FUNCTION_BLOCK "Blok_Pracy_Bindownicy"	// FB 35
//Funkcja odpowiada za sterowanie calym procesem bindowania
//Jezeli dane zostaly zmienione w trakcie trwania cyklu to dopiero w czasie 
//nowego 
//cyklu zostana przyjete.
//
//
//
VERSION : 0.1
VAR_INPUT
  i_Marka_Bezpieczenstwa : BOOL ;
  i_Auto_Reczny : BOOL ;
  i_Bindownica_Auto : BOOL ;
  i_Start_Cyklu_Auto : BOOL ;
  i_Reset_Bledu_Cyklu : BOOL ;
  i_Reset_Cyklu : BOOL ;	//Sprowadza funkcje do poczatku
  i_Pozycjonuj_Palete : BOOL ;
  i_TP_Wiazanie_0_st : BOOL ;
  i_TP_Wiazanie_90_st : BOOL ;
  i_TP_Wiazanie_180_st : BOOL ;
  i_TP_Wiazanie_270_st : BOOL ;
  i_TP_Pozycjonowanie : BOOL ;
  i_s_Zez_Rolki : BOOL ;
  i_Pozycja_Bandy_Lewo : BOOL ;
  i_Pozycja_Bandy_Srodek : BOOL ;
  i_Pozycja_Bandy_Prawo : BOOL ;
  i_Pozycja_Bandy_Potw : BOOL ;
  i_Pozycja_Obr_0st : BOOL ;
  i_Pozycja_Obr_90st : BOOL ;
  i_Pozycja_Obr_180st : BOOL ;
  i_Pozycja_Obr_270st : BOOL ;
  i_Pozycja_Obr_Osiagnieta : BOOL ;
  i_Bind_Obwod_Ok : BOOL ;
  i_Bind_Poloz_Podst : BOOL ;
  i_Bind_Start_Kon_Wiaz : BOOL ;
  i_Bind_Blad : BOOL ;
  i_Wyjazd_Warunkowy : BOOL ;
  i_Fotokomorki_Pokryte : BOOL ;
  i_Start_Cyklu_Reczny : BOOL ;
  i_Rezerwa_4 : BOOL ;
  i_Rezerwa_5 : BOOL ;
END_VAR
VAR_OUTPUT
  o_Pozycjonuj_Lewo : BOOL ;
  o_Pozycjonuj_Prawo : BOOL ;
  o_Pozycjonuj_Srodek : BOOL ;
  o_Jedz_Na_0st : BOOL ;
  o_Jedz_Na_90st : BOOL ;
  o_Jedz_Na_180st : BOOL ;
  o_Jedz_Na_270st : BOOL ;
  o_Bind_Zez_Na_Prace : BOOL ;
  o_Bind_Start_Wiazan : BOOL ;
  o_Koniec_Cyklu : BOOL ;
  o_Cykl_W_Trakcie : BOOL ;	//informacja ze maszyna jest w trakcie cyklu
  o_Blad_Ogolny : BOOL ;
  o_Blad_Cyklu : BOOL ;
  o_Rezerwa_1 : BOOL ;
  o_Rezerwa_2 : BOOL ;
  o_Rezerwa_3 : BOOL ;
  o_Rezerwa_4 : BOOL ;
END_VAR
VAR_IN_OUT
  io_Step_Counter : INT ;
END_VAR
VAR
  Kontrola_Tranzycji : FB 20;	//Timmer kontrolujacy czy krok jest konczony
  Timer_Pauzy : FB 20;
  Timer_Kon_Strzalu : FB 20;	//Timer kontroli strzalu
  Tim_Rezerwa_2 : FB 20;
  Tim_Rezerwa_3 : FB 20;
  H_Czas_Kontrolny : TIME ;
  Stop_Czas_Kontrolny : BOOL ;
  H_Czas_Pauzy : TIME ;
  Start_Bindowania : BOOL ;
  H_Obr_Na_Poz_X : BOOL ;
  H_Pozycjonuj_Srodek : BOOL ;
  H_Pozycjonuj_Lewo : BOOL ;
  H_Pozycjonuj_Prawo : BOOL ;
  H_Wykonaj_Wiazanie : BOOL ;
  H_Wiazanie_Zak_Pom : BOOL ;
  H_Jedz_Na_Poz_X : BOOL ;
  H_Paleta_Na_Prawo : BOOL ;
  H_Paleta_Na_Srodku : BOOL ;
  H_Paleta_Na_Lewo : BOOL ;
  H_Wiazanie_0_st : BOOL ;
  H_Wiazanie_90_st : BOOL ;
  H_Wiazanie_180_st : BOOL ;
  H_Wiazanie_270_st : BOOL ;
  H_Pozycjonowanie : BOOL ;
  H_Blad : BOOL ;
  Bit_Tranzycji : BOOL ;
  Zbocze_1 : BOOL ;
  H_Bit_Pauzy : BOOL ;
  H_Poczatek_Pauzy : BOOL ;
  H_Koniec_Pauzy : BOOL ;
  Krok_1 : BOOL ;
  Krok_2 : BOOL ;
  Krok_3 : BOOL ;
  Krok_4 : BOOL ;
  Krok_5 : BOOL ;
  Krok_6 : BOOL ;
  Krok_7 : BOOL ;
  Krok_8 : BOOL ;
  Krok_9 : BOOL ;
  Trwa_Krok_1 : BOOL ;
  Trwa_Krok_2 : BOOL ;
  Trwa_Krok_3 : BOOL ;
  Trwa_Krok_4 : BOOL ;
  Trwa_Krok_5 : BOOL ;
  Trwa_Krok_6 : BOOL ;
  Trwa_Krok_7 : BOOL ;
  Trwa_Krok_8 : BOOL ;
  Trwa_Krok_9 : BOOL ;
  Zadanie_1 : BOOL ;
  Zadanie_2 : BOOL ;
  Zadanie_3 : BOOL ;
  Zadanie_4 : BOOL ;
  Zadanie_5 : BOOL ;
  Zadanie_6 : BOOL ;
  Zadanie_10 : BOOL ;
  H_int : INT ;
  H_Pozycja_0_st_ok : BOOL ;
  H_Pozycja_90_st_ok : BOOL ;
  H_Pozycja_180_st_ok : BOOL ;
  H_Pozycja_270_st_ok : BOOL ;
  Zbocze_2 : BOOL ;
  H_Bindownic_Skon_Wiaz : BOOL ;
  H_19 : BOOL ;
  H_20 : BOOL ;
  H_30 : BOOL ;
  H_31 : BOOL ;
  H_32 : BOOL ;
  H_22 : BOOL ;
  H_34 : BOOL ;
  H_45 : BOOL ;
  H_23 : BOOL ;
END_VAR
VAR_TEMP
  Help_Bit_1 : BOOL ;
  Help_Bit_2 : BOOL ;
  Bit_Kontroli_Czasu : BOOL ;
  Czas_Aktualny : TIME ;
  Help_Bit_3 : BOOL ;
END_VAR
BEGIN
NETWORK
TITLE =
//Ten network celow jest wolny
//
NETWORK
TITLE =
//Przygotowanie marki bezpieczenstw
      A     #i_Marka_Bezpieczenstwa;
      S     #Stop_Czas_Kontrolny;
      AN    #i_Marka_Bezpieczenstwa;
      R     #Stop_Czas_Kontrolny;
NETWORK
TITLE =
//Przygotowanie do startu
//
//
//********************************************
//Reset konca cyklu
      L     0;
      L     #io_Step_Counter;
      ==I;
      R     #o_Koniec_Cyklu;
//********************************************
//Rozpoczecie bindowania
      A     #o_Koniec_Cyklu;
      JCN   et_1;
      L     0;
      T     #io_Step_Counter;
et_1: NOP   0;
//********************************************
// Start cyklu bindowania
      A     #i_Auto_Reczny;
      A     #i_Start_Cyklu_Auto;
      AN    #o_Cykl_W_Trakcie;
      O;
      A     #i_Start_Cyklu_Reczny;
      AN    #i_Auto_Reczny;
      AN    #o_Cykl_W_Trakcie;
      S     #Start_Bindowania;
//********************************************
//Zresetowanie bitow startowych
      A     #i_Auto_Reczny;
      A     #Start_Bindowania;
      JCN   et_a;
      L     2;
      T     #io_Step_Counter;
      SET;
      R     #Start_Bindowania;
et_a: NOP   0;
      AN    #i_Auto_Reczny;
      A     #Start_Bindowania;
      JCN   et_r;
      L     1;
      T     #io_Step_Counter;
      SET;
      R     #Start_Bindowania;
et_r: NOP   0;
//********************************************
//Gdy reset wcisniety to kasuj wszystkie bity
      AN    #i_Auto_Reczny;
      A     #i_Reset_Cyklu;
      JCN   et_3;
      L     0;
      T     #io_Step_Counter;
      SET;
      R     #o_Koniec_Cyklu;
      R     #o_Cykl_W_Trakcie;
      JU    clrs;
et_3: NOP   0;
//********************************************
//Pozycjonowanie palety
      A     #i_Pozycjonuj_Palete;
      JCN   et_4;
      L     10;
      T     #io_Step_Counter;
et_4: NOP   0;
//********************************************
//Maszyna w trakcie cyklu bindowania
      L     #io_Step_Counter;
      L     0;
      <>I;
      =     #o_Cykl_W_Trakcie;
//********************************************
//Przypisanie jazdy do nowych pozycji gdy koniec cyklu
      A     #o_Cykl_W_Trakcie;
      JC    et_5;
//0st
      A     #i_TP_Wiazanie_0_st;
      =     #H_Wiazanie_0_st;
//90st
      A     #i_TP_Wiazanie_90_st;
      =     #H_Wiazanie_90_st;
//180st
      A     #i_TP_Wiazanie_180_st;
      =     #H_Wiazanie_180_st;
//270st
      A     #i_TP_Wiazanie_270_st;
      =     #H_Wiazanie_270_st;
//Pozycjonowanie
      A     #i_TP_Pozycjonowanie;
      =     #H_Pozycjonowanie;
et_5: NOP   0;
//********************************************
//Wyjazd warunkowy
      A     #i_Pozycja_Obr_0st;
      A     #i_Auto_Reczny;
      A     #i_Wyjazd_Warunkowy;
      AN    #o_Cykl_W_Trakcie;
      JCN   et_6;
      L     6;
      T     #io_Step_Counter;
et_6: NOP   0;
NETWORK
TITLE =
//Lista Zadan Pracy
//
//**************Zadania  ***********************
//Srodkowanie dla 0 
      L     #io_Step_Counter;
      L     1;
      ==I;
      =     #Zadanie_1;
//0st
      L     #io_Step_Counter;
      L     2;
      ==I;
      =     #Zadanie_2;
//90st
      L     #io_Step_Counter;
      L     3;
      ==I;
      =     #Zadanie_3;
//180st
      L     #io_Step_Counter;
      L     4;
      ==I;
      =     #Zadanie_4;
//270st
      L     #io_Step_Counter;
      L     5;
      ==I;
      =     #Zadanie_5;
//powrot 0st
      L     #io_Step_Counter;
      L     6;
      ==I;
      =     #Zadanie_6;
//reset
      L     #io_Step_Counter;
      L     10;
      ==I;
      =     #Zadanie_10;
NETWORK
TITLE =
//Maszyna z krokiem nr 0
//Jezeli wartosc licznika 0 to
//Wyczysc wszystko i wyjdz
      L     #io_Step_Counter;
      L     0;
      ==I;
      JC    clrs;
NETWORK
TITLE =
//Zadanie nr 1 srodkuj palete Wersja dzialajaca:   
//       A     #Zadanie_1
//      JCN   u_1
//
//      SET   
//      S     #Krok_1
////***************************************************
////Krok 1 - jedz na pozycje 0st 
//
//      A     #Krok_1
//      AN    #Krok_2
//      R     #H_Paleta_Na_Srodku
//
//
//
//      A     #H_Obr_Na_Poz_X
//      S     #Krok_2
//      R     #H_Obr_Na_Poz_X
//      R     #H_Jedz_Na_Poz_X
////-
//      A     #Krok_1
//      AN    #Krok_2
//      =     #Trwa_Krok_1
//      S     #H_Jedz_Na_Poz_X
//      JC    j_1
//
////***************************************************
////Krok 2 - Jezeli tryb z pozycjonowaniem to wyœrodkuj palete
//
//
//
//      A     #H_Paleta_Na_Srodku
//      AN    #Krok_3
//      S     #Krok_3
//      R     #H_Pozycjonuj_Srodek
//      R     #H_Paleta_Na_Srodku
////-
//      A     #Krok_2
//      AN    #Krok_3
//      =     #Trwa_Krok_2
//      S     #H_Pozycjonuj_Srodek
//      JC    res
//
//
////Krok 3 - Przejscie do kroku inkrementu
//
//      A     #Krok_3
//      S     #Krok_7
//
////Krok 7 - Zadanie ukonczone przejdz do nastepnego zadania
//
//      A     #Krok_7
//      JC    inc
//
//u_1:  NOP   0
//
      A     #Zadanie_1;
      JCN   u_1;
      SET;
      S     #Krok_1;
//***************************************************
//Krok 1 - jedz na pozycje 0st 
      A     #Krok_1;
      AN    #Krok_2;
      R     #H_Paleta_Na_Srodku;
      A     #Krok_1;
      A(;
      O     #i_Pozycja_Obr_0st;
      O     #i_Pozycja_Obr_180st;
      );
      S     #Krok_2;
//****************************************************
//jezeli nie ma pozycji to wyzeruj
      AN    #Krok_2;
      JC    zer;
//****************************************************
//Krok 2 - Jezeli tryb z pozycjonowaniem to wysrodkuj palete
      A     #H_Paleta_Na_Srodku;
      AN    #Krok_3;
      S     #Krok_3;
      R     #H_Pozycjonuj_Srodek;
      R     #H_Paleta_Na_Srodku;
//-
      A     #Krok_2;
      AN    #Krok_3;
      =     #Trwa_Krok_2;
      S     #H_Pozycjonuj_Srodek;
      JC    res;
//Krok 3 - Przejscie do kroku inkrementu
      A     #Krok_3;
      S     #Krok_7;
//Krok 7 - Zadanie ukonczone przejdz do nastepnego zadania
      A     #Krok_7;
      JC    inc;
u_1:  NOP   0;
NETWORK
TITLE =
//Zadanie nr 2 wiazanie na pozycji 0st
//**************Zadanie 2 ***********************
      A     #Zadanie_2;
      JCN   u_2;
//***************************************************
//Wyskocz jezeli brak wiazania dla 0st
      AN    #H_Wiazanie_0_st;
      JC    inc;
//***************************************************
//Rozpoczecie grafu
      SET;
      S     #Krok_1;
//***************************************************
//Krok 1 - jedz na pozycje 0st 
      A     #H_Obr_Na_Poz_X;
      S     #Krok_2;
      R     #H_Obr_Na_Poz_X;
      R     #H_Jedz_Na_Poz_X;
//-
      A     #Krok_1;
      AN    #Krok_2;
      =     #Trwa_Krok_1;
      S     #H_Jedz_Na_Poz_X;
      JC    j_1;
//***************************************************
//Krok 2 - Jezeli tryb z pozycjonowaniem to wyœrodkuj palete
      A     #H_Pozycjonowanie;
      A     #H_Paleta_Na_Srodku;
      AN    #Krok_3;
      O;
      AN    #H_Pozycjonowanie;
      AN    #Krok_3;
      S     #Krok_3;
      R     #H_Pozycjonuj_Srodek;
      R     #H_Paleta_Na_Srodku;
//-
      A     #Krok_2;
      AN    #Krok_3;
      =     #Trwa_Krok_2;
      S     #H_Pozycjonuj_Srodek;
      JC    res;
//***************************************************
//Krok 3 - Dla 0 stopni pozycjonuj w prawo przed strza³em
      A     #H_Pozycjonowanie;
      A     #H_Paleta_Na_Prawo;
      O;
      AN    #H_Pozycjonowanie;
      S     #Krok_4;
      R     #H_Pozycjonuj_Prawo;
      R     #H_Paleta_Na_Prawo;
//-
      A     #Krok_3;
      AN    #Krok_4;
      =     #Trwa_Krok_3;
      S     #H_Pozycjonuj_Prawo;
      JC    pp;
//***************************************************
//Krok 4 -Wykonaj wiazanie
      A     #H_Wiazanie_Zak_Pom;
      S     #Krok_5;
      R     #H_Wykonaj_Wiazanie;
      R     #H_Wiazanie_Zak_Pom;
      R     #H_Bindownic_Skon_Wiaz;
//-
      A     #Krok_4;
      AN    #Krok_5;
      =     #Trwa_Krok_4;
      S     #H_Wykonaj_Wiazanie;
      JC    bind;
//*****************************************************
//Krok 5 - Przerwa po zwiazaniu
      A     #H_Koniec_Pauzy;
      S     #Krok_6;
      R     #H_Poczatek_Pauzy;
      R     #H_Koniec_Pauzy;
//-
      L     T#2S;
      T     #H_Czas_Pauzy;
//-
      A     #Krok_5;
      AN    #Krok_6;
      =     #Trwa_Krok_5;
      S     #H_Poczatek_Pauzy;
      JC    wait;
//*****************************************************
//Krok 6 - Jezeli tryb z pozycjonowaniem to wyœrodkuj palete
      A     #H_Pozycjonowanie;
      A     #H_Paleta_Na_Srodku;
      AN    #Krok_7;
      O;
      AN    #H_Pozycjonowanie;
      AN    #Krok_7;
      S     #Krok_7;
      R     #H_Pozycjonuj_Srodek;
      R     #H_Paleta_Na_Srodku;
//-
      A     #Krok_6;
      AN    #Krok_7;
      =     #Trwa_Krok_6;
      S     #H_Pozycjonuj_Srodek;
      JC    res;
//***************************************************
//Krok 7 - Zadanie ukonczone przejdz do nastepnego zadania
      A     #Krok_7;
      JC    inc;
u_2:  NOP   0;
NETWORK
TITLE =
//Zadanie nr 3 wiazanie na pozycji 90st
//**************Zadanie 3 ***********************
      A     #Zadanie_3;
      JCN   u_3;
//***************************************************
//Wyskocz jezeli brak wiazania dla 0st
      AN    #H_Wiazanie_90_st;
      JC    inc;
//***************************************************
//Rozpoczecie grafu
      SET;
      S     #Krok_1;
//***************************************************
//Krok 1 - jedz na pozycje 90st 
      A     #H_Obr_Na_Poz_X;
      S     #Krok_2;
      R     #H_Obr_Na_Poz_X;
      R     #H_Jedz_Na_Poz_X;
//-
      A     #Krok_1;
      AN    #Krok_2;
      =     #Trwa_Krok_1;
      S     #H_Jedz_Na_Poz_X;
      JC    j_2;
//***************************************************
//Przejdz pominiete kroki
      A     #Krok_2;
      S     #Krok_3;
//-
      A     #Krok_3;
      S     #Krok_4;
//***************************************************
//Krok 4 -Wykonaj wiazanie
      A     #H_Wiazanie_Zak_Pom;
      S     #Krok_5;
      R     #H_Wykonaj_Wiazanie;
      R     #H_Wiazanie_Zak_Pom;
      R     #H_Bindownic_Skon_Wiaz;
//-
      A     #Krok_4;
      AN    #Krok_5;
      =     #Trwa_Krok_4;
      S     #H_Wykonaj_Wiazanie;
      JC    bind;
//*****************************************************
//Krok 5 - Przerwa po zwiazaniu
      A     #H_Koniec_Pauzy;
      S     #Krok_6;
      R     #H_Poczatek_Pauzy;
      R     #H_Koniec_Pauzy;
//-
      L     T#2S;
      T     #H_Czas_Pauzy;
//-
      A     #Krok_5;
      AN    #Krok_6;
      =     #Trwa_Krok_5;
      S     #H_Poczatek_Pauzy;
      JC    wait;
//*****************************************************
//Krok 6
      A     #Krok_6;
      S     #Krok_7;
//***************************************************
//Krok 7 - Zadanie ukonczone przejdz do nastepnego zadania
      A     #Krok_7;
      JC    inc;
u_3:  NOP   0;
NETWORK
TITLE =
//Zadanie nr 4 wiazanie na pozycji 180st
//**************Zadanie 4 ***********************
      A     #Zadanie_4;
      JCN   u_4;
//***************************************************
//Wyskocz jezeli brak wiazania dla 0st
      AN    #H_Wiazanie_180_st;
      JC    inc;
//***************************************************
//Rozpoczecie grafu
      SET;
      S     #Krok_1;
//***************************************************
//Krok 1 - jedz na pozycje 0st 
      A     #H_Obr_Na_Poz_X;
      S     #Krok_2;
      R     #H_Obr_Na_Poz_X;
      R     #H_Jedz_Na_Poz_X;
//-
      A     #Krok_1;
      AN    #Krok_2;
      =     #Trwa_Krok_1;
      S     #H_Jedz_Na_Poz_X;
      JC    j_3;
//***************************************************
//Krok 2 - Jezeli tryb z pozycjonowaniem to wyœrodkuj palete
      A     #H_Pozycjonowanie;
      A     #H_Paleta_Na_Srodku;
      AN    #Krok_3;
      O;
      AN    #H_Pozycjonowanie;
      AN    #Krok_3;
      S     #Krok_3;
      R     #H_Pozycjonuj_Srodek;
      R     #H_Paleta_Na_Srodku;
//-
      A     #Krok_2;
      AN    #Krok_3;
      =     #Trwa_Krok_2;
      S     #H_Pozycjonuj_Srodek;
      JC    res;
//***************************************************
//Krok 3 - Dla 180 stopni pozycjonuj w lewo przed strza³em
      A     #H_Pozycjonowanie;
      A     #H_Paleta_Na_Lewo;
      O;
      AN    #H_Pozycjonowanie;
      S     #Krok_4;
      R     #H_Pozycjonuj_Lewo;
      R     #H_Paleta_Na_Lewo;
//-
      A     #Krok_3;
      AN    #Krok_4;
      =     #Trwa_Krok_3;
      S     #H_Pozycjonuj_Lewo;
      JC    pl;
//***************************************************
//Krok 4 -Wykonaj wiazanie
      A     #H_Wiazanie_Zak_Pom;
      S     #Krok_5;
      R     #H_Wykonaj_Wiazanie;
      R     #H_Wiazanie_Zak_Pom;
      R     #H_Bindownic_Skon_Wiaz;
//-
      A     #Krok_4;
      AN    #Krok_5;
      =     #Trwa_Krok_4;
      S     #H_Wykonaj_Wiazanie;
      JC    bind;
//*****************************************************
//Krok 5 - Przerwa po zwiazaniu
      A     #H_Koniec_Pauzy;
      S     #Krok_6;
      R     #H_Poczatek_Pauzy;
      R     #H_Koniec_Pauzy;
//-
      L     T#2S;
      T     #H_Czas_Pauzy;
//-
      A     #Krok_5;
      AN    #Krok_6;
      =     #Trwa_Krok_5;
      S     #H_Poczatek_Pauzy;
      JC    wait;
//*****************************************************
//Krok 6 - Jezeli tryb z pozycjonowaniem to wyœrodkuj palete
      A     #H_Pozycjonowanie;
      A     #H_Paleta_Na_Srodku;
      AN    #Krok_7;
      O;
      AN    #H_Pozycjonowanie;
      AN    #Krok_7;
      S     #Krok_7;
      R     #H_Pozycjonuj_Srodek;
      R     #H_Paleta_Na_Srodku;
//-
      A     #Krok_6;
      AN    #Krok_7;
      =     #Trwa_Krok_6;
      S     #H_Pozycjonuj_Srodek;
      JC    res;
//***************************************************
//Krok 7 - Zadanie ukonczone przejdz do nastepnego zadania
      A     #Krok_7;
      JC    inc;
u_4:  NOP   0;
NETWORK
TITLE =
//Zadanie nr 3 wiazanie na pozycji 270st
//**************Zadanie 5 ***********************
      A     #Zadanie_5;
      JCN   u_5;
//***************************************************
//Wyskocz jezeli brak wiazania dla 0st
      AN    #H_Wiazanie_270_st;
      JC    inc;
//***************************************************
//Rozpoczecie grafu
      SET;
      S     #Krok_1;
//***************************************************
//Krok 1 - jedz na pozycje 90st 
      A     #H_Obr_Na_Poz_X;
      S     #Krok_2;
      R     #H_Obr_Na_Poz_X;
      R     #H_Jedz_Na_Poz_X;
//-
      A     #Krok_1;
      AN    #Krok_2;
      =     #Trwa_Krok_1;
      S     #H_Jedz_Na_Poz_X;
      JC    j_4;
//***************************************************
//Przejdz pominiete kroki
      A     #Krok_2;
      S     #Krok_3;
//-
      A     #Krok_3;
      S     #Krok_4;
//***************************************************
//Krok 4 -Wykonaj wiazanie
      A     #H_Wiazanie_Zak_Pom;
      S     #Krok_5;
      R     #H_Wykonaj_Wiazanie;
      R     #H_Wiazanie_Zak_Pom;
      R     #H_Bindownic_Skon_Wiaz;
//-
      A     #Krok_4;
      AN    #Krok_5;
      =     #Trwa_Krok_4;
      S     #H_Wykonaj_Wiazanie;
      JC    bind;
//*****************************************************
//Krok 5 - Przerwa po zwiazaniu
      A     #H_Koniec_Pauzy;
      S     #Krok_6;
      R     #H_Poczatek_Pauzy;
      R     #H_Koniec_Pauzy;
//-
      L     T#2S;
      T     #H_Czas_Pauzy;
//-
      A     #Krok_5;
      AN    #Krok_6;
      =     #Trwa_Krok_5;
      S     #H_Poczatek_Pauzy;
      JC    wait;
//*****************************************************
//Krok 6
      A     #Krok_6;
      S     #Krok_7;
//***************************************************
//Krok 7 - Zadanie ukonczone przejdz do nastepnego zadania
      A     #Krok_7;
      JC    inc;
u_5:  NOP   0;
NETWORK
TITLE =
//Zadanie nr 6 Powrot do pozycji wyjazdu
//**************Zadanie 6 ***********************
      A     #Zadanie_6;
      JCN   u_6;
//Rozpoczecie grafu
      SET;
      S     #Krok_1;
//***************************************************
//Krok 1 - jedz na pozycje 0st 
      A     #H_Obr_Na_Poz_X;
      S     #Krok_2;
      R     #H_Obr_Na_Poz_X;
      R     #H_Jedz_Na_Poz_X;
//-
      A     #Krok_1;
      AN    #Krok_2;
      =     #Trwa_Krok_1;
      S     #H_Jedz_Na_Poz_X;
      JC    j_1;
//Pozkaz ze koniec cyklu
      A     #Krok_2;
      S     #Krok_8;
      A     #Krok_8;
      S     #o_Koniec_Cyklu;
      JC    clrs;
u_6:  NOP   0;
NETWORK
TITLE =
//Zadanie wyzerowania palety na obrotnicy
//**************Zadanie 10 ***********************
      A     #Zadanie_10;
      JCN   u_10;
//***************************************************
//Rozpoczecie grafu
      SET;
      S     #Krok_1;
//***************************************************
//Krok 1 - jedz na pozycje 0st 
      A     #H_Obr_Na_Poz_X;
      S     #Krok_2;
      R     #H_Obr_Na_Poz_X;
      R     #H_Jedz_Na_Poz_X;
//-
      A     #Krok_1;
      AN    #Krok_2;
      =     #Trwa_Krok_1;
      S     #H_Jedz_Na_Poz_X;
      JC    j_1;
//***************************************************
//Krok 2 - Jezeli tryb z pozycjonowaniem to wyœrodkuj palete
      A     #H_Paleta_Na_Srodku;
      O;
      S     #Krok_3;
      R     #H_Pozycjonuj_Srodek;
      R     #H_Paleta_Na_Srodku;
//-
      A     #Krok_2;
      AN    #Krok_3;
      =     #Trwa_Krok_2;
      S     #H_Pozycjonuj_Srodek;
      JC    res;
//-
      L     0;
      T     #io_Step_Counter;
      JU    clrs;
u_10: NOP   0;
      JU    tim;
NETWORK
TITLE =
//Puste celowo
NETWORK
TITLE =
//Rozkazy do maszyny bindujacej 
// bindowanie 
bind: NOP   0;
      A     #H_Wykonaj_Wiazanie;
      AN    #o_Bind_Start_Wiazan;
      R     #H_Bindownic_Skon_Wiaz;
      =     #H_19;
      A     #H_Wykonaj_Wiazanie;
      A     #i_Fotokomorki_Pokryte;
      S     #o_Bind_Start_Wiazan;
      A     #i_Bind_Start_Kon_Wiaz;
      FP    #Zbocze_1;
      S     #H_Wiazanie_Zak_Pom;
      R     #H_Wykonaj_Wiazanie;
      R     #o_Bind_Start_Wiazan;
      R     #Bit_Tranzycji;
      R     #H_Bindownic_Skon_Wiaz;
//bindownica wraca
      A     #i_Bind_Poloz_Podst;
      FP    #Zbocze_2;
      A     #o_Bind_Start_Wiazan;
      AN    #H_19;
      S     #H_Bindownic_Skon_Wiaz;
      A     #o_Bind_Start_Wiazan;
      A     #i_Bindownica_Auto;
      A     #H_Bindownic_Skon_Wiaz;
      AN    #H_19;
      =     #Help_Bit_1;
      CALL  #Timer_Kon_Strzalu (
           IN                       := #Help_Bit_1,
           STOP                     := #Stop_Czas_Kontrolny,
           PT                       := T#3S,
           Q_0                      := #Help_Bit_2,
           ET                       := #Czas_Aktualny);
      A     #Help_Bit_2;
      S     #H_Wiazanie_Zak_Pom;
      R     #H_Wykonaj_Wiazanie;
      R     #o_Bind_Start_Wiazan;
      R     #Bit_Tranzycji;
      R     #H_Bindownic_Skon_Wiaz;
      JU    tim;
//Pozycjonowanie Prawo
pp:   NOP   0;
      A     #H_Pozycjonuj_Prawo;
      S     #o_Pozycjonuj_Prawo;
//-
      A     #i_Pozycja_Bandy_Prawo;
      A     #i_Pozycja_Bandy_Potw;
      S     #H_Paleta_Na_Prawo;
      R     #H_Pozycjonuj_Prawo;
      R     #o_Pozycjonuj_Prawo;
      R     #Bit_Tranzycji;
      JU    tim;
//Pozycjonowanie lewo
pl:   NOP   0;
      A     #H_Pozycjonuj_Lewo;
      S     #o_Pozycjonuj_Lewo;
//-
      A     #i_Pozycja_Bandy_Lewo;
      A     #i_Pozycja_Bandy_Potw;
      S     #H_Paleta_Na_Lewo;
      R     #H_Pozycjonuj_Lewo;
      R     #o_Pozycjonuj_Lewo;
      R     #Bit_Tranzycji;
      JU    tim;
//resetowanie pozycjonowania
res:  NOP   0;
      A     #H_Pozycjonuj_Srodek;
      S     #o_Pozycjonuj_Srodek;
//-
      A     #i_Pozycja_Bandy_Srodek;
      A     #i_Pozycja_Bandy_Potw;
      S     #H_Paleta_Na_Srodku;
      R     #H_Pozycjonuj_Srodek;
      R     #o_Pozycjonuj_Srodek;
      R     #Bit_Tranzycji;
      JU    tim;
//osiagniecie pozycji 270st
j_4:  NOP   0;
      A     #H_Jedz_Na_Poz_X;
      S     #o_Jedz_Na_270st;
      A     #i_Pozycja_Obr_270st;
      A     #i_Pozycja_Obr_Osiagnieta;
      S     #H_Obr_Na_Poz_X;
      R     #o_Jedz_Na_270st;
      R     #H_Jedz_Na_Poz_X;
      R     #Bit_Tranzycji;
      JU    tim;
//osiagniecie pozycji 180st
j_3:  NOP   0;
      A     #H_Jedz_Na_Poz_X;
      S     #o_Jedz_Na_180st;
      A     #i_Pozycja_Obr_180st;
      A     #i_Pozycja_Obr_Osiagnieta;
      S     #H_Obr_Na_Poz_X;
      R     #o_Jedz_Na_180st;
      R     #H_Jedz_Na_Poz_X;
      R     #Bit_Tranzycji;
      JU    tim;
//osiagniecie pozycji 90st
j_2:  NOP   0;
      A     #H_Jedz_Na_Poz_X;
      S     #o_Jedz_Na_90st;
      A     #i_Pozycja_Obr_90st;
      A     #i_Pozycja_Obr_Osiagnieta;
      S     #H_Obr_Na_Poz_X;
      R     #o_Jedz_Na_90st;
      R     #H_Jedz_Na_Poz_X;
      R     #Bit_Tranzycji;
      JU    tim;
//osiagniecie pozycji 0st
j_1:  NOP   0;
      A     #H_Jedz_Na_Poz_X;
      S     #o_Jedz_Na_0st;
      A     #i_Pozycja_Obr_0st;
      A     #i_Pozycja_Obr_Osiagnieta;
      S     #H_Obr_Na_Poz_X;
      R     #o_Jedz_Na_0st;
      R     #H_Jedz_Na_Poz_X;
      R     #Bit_Tranzycji;
      JU    tim;
//zerowanie licznika
zer:  NOP   0;
      L     0;
      T     #io_Step_Counter;
      JU    clrs;
//Zwiekszenie licznika krokow o 1  
inc:  NOP   0;
      L     #io_Step_Counter;
      L     1;
      +I;
      T     #io_Step_Counter;
clrs: SET;
//resetowanie bitow pracy programu
//k1
      R     #H_Jedz_Na_Poz_X;
      R     #H_Obr_Na_Poz_X;
//k2
      R     #H_Pozycjonuj_Srodek;
      R     #H_Paleta_Na_Srodku;
//k3
      R     #H_Pozycjonuj_Prawo;
      R     #H_Paleta_Na_Prawo;
//k4
      R     #H_Pozycjonuj_Lewo;
      R     #H_Paleta_Na_Lewo;
//k5
      R     #H_Wykonaj_Wiazanie;
      R     #H_Wiazanie_Zak_Pom;
      R     #H_Wykonaj_Wiazanie;
      R     #H_Bindownic_Skon_Wiaz;
      R     #H_Wiazanie_Zak_Pom;
//k6
      R     #H_Poczatek_Pauzy;
      R     #H_Koniec_Pauzy;
      R     #H_Bit_Pauzy;
//Bt
      R     #Bit_Tranzycji;
      R     #H_Bindownic_Skon_Wiaz;
//-
      R     #Krok_1;
      R     #Krok_2;
      R     #Krok_3;
      R     #Krok_4;
      R     #Krok_5;
      R     #Krok_6;
      R     #Krok_7;
      R     #Krok_8;
      R     #Krok_9;
//-
      R     #Trwa_Krok_1;
      R     #Trwa_Krok_2;
      R     #Trwa_Krok_3;
      R     #Trwa_Krok_4;
      R     #Trwa_Krok_5;
      R     #Trwa_Krok_6;
      R     #Trwa_Krok_7;
      R     #Trwa_Krok_8;
      R     #Trwa_Krok_9;
//-
      R     #o_Pozycjonuj_Lewo;
      R     #o_Pozycjonuj_Prawo;
      R     #o_Pozycjonuj_Srodek;
      R     #o_Jedz_Na_0st;
      R     #o_Jedz_Na_90st;
      R     #o_Jedz_Na_180st;
      R     #o_Jedz_Na_270st;
      R     #o_Bind_Start_Wiazan;
//      R     #Zbocze_2
//      R     #Zbocze_1
      JU    tim;
//Czas Pauzy
wait: NOP   0;
      CALL  #Timer_Pauzy (
           IN                       := #H_Bit_Pauzy,
           STOP                     := #Stop_Czas_Kontrolny,
           PT                       := #H_Czas_Pauzy,
           Q_0                      := #Help_Bit_1,
           ET                       := #Czas_Aktualny);
      A     #H_Poczatek_Pauzy;
      S     #H_Bit_Pauzy;
      A     #Help_Bit_1;
      R     #H_Poczatek_Pauzy;
      R     #H_Bit_Pauzy;
      S     #H_Koniec_Pauzy;
      JU    tim;
NETWORK
TITLE =
//Czas kontrolny poszczegolnych krokow
//**************************************************
//Kontynuacja programu sprawdzenie czasow tranzycji
tim:  NOP   0;
//**************************************************
//Sprawdzenie ktory krok jest aktywny 
      O     #Zadanie_1;
      O     #Zadanie_2;
      O     #Zadanie_3;
      O     #Zadanie_4;
      O     #Zadanie_5;
      O     #Zadanie_10;
      JCN   z_1;
//krok_1  - jedz na pozycje 
      A     #Trwa_Krok_1;
      =     "Blok_Para".Krok_1;
      L     T#20S;
      JC    z_2;
//krok_2 - szukaj srodka 
      A     #Trwa_Krok_2;
      L     T#10S;
      =     "Blok_Para".krok_2;
      JC    z_2;
//krok_3 - jedz na prawo
      A     #Trwa_Krok_3;
      L     T#10S;
      =     "Blok_Para".krok_3;
      JC    z_2;
//krok_4 - strzelaj 
      A     #Trwa_Krok_4;
      L     T#2M;
      =     "Blok_Para".krok_4;
      JC    z_2;
//krok_5  - pauza po strzale
      A     #Trwa_Krok_5;
      L     T#10S;
      =     "Blok_Para".krok_5;
      JC    z_2;
//krok_6 - jedz do srodka
      A     #Trwa_Krok_6;
      L     T#10S;
      =     "Blok_Para".krok_6;
      JC    z_2;
z_1:  NOP   0;
NETWORK
TITLE =
NETWORK
TITLE =
//Sprawdzenie czy czas nie przeszedl za daleko
//Zaladuj czas oraz wystartuj timmer
//koniec kazdego z krokow resetuje timmer
z_2:  SET;
      =     #Help_Bit_1;
      T     #H_Czas_Kontrolny;
//-  
      A     "Zawsze_False";
      A     #Help_Bit_1;
      A     #Bit_Tranzycji;
      =     #Help_Bit_2;
      CALL  #Kontrola_Tranzycji (
           IN                       := #Help_Bit_2,
           STOP                     := #Stop_Czas_Kontrolny,
           PT                       := #H_Czas_Kontrolny,
           Q_0                      := #Help_Bit_3,
           ET                       := #Czas_Aktualny);
      SET;
      S     #Bit_Tranzycji;
//Blad czasu tranzycji maszyna nie przeszla do 
//dalszego kroku
      SET;
      R     #H_Blad;
      A     "Zawsze_False";
      A     #Help_Bit_3;
      S     #H_Blad;
NETWORK
TITLE = Blad kroku nr 1 (Przekrokczony czas jazdy  na zadana pozycje)
//Zbuduj kod beledu
//kod bledu to nr licznika oraz
//nr kroku
//lista bledow
      A     #H_Blad;
      =     #o_Blad_Cyklu;
      A     #i_Reset_Bledu_Cyklu;
      R     #H_Blad;
      A     #H_Blad;
      A     #Trwa_Krok_1;
      S     "Blok_Bledow_Program".Blad_Krok_1;
      A     #H_Blad;
      A     #Trwa_Krok_2;
      S     "Blok_Bledow_Program".Blad_Krok_2;
      A     #H_Blad;
      A     #Trwa_Krok_3;
      S     "Blok_Bledow_Program".Blad_Krok_3;
      A     #H_Blad;
      A     #Trwa_Krok_4;
      S     "Blok_Bledow_Program".Blad_Krok_4;
      A     #H_Blad;
      A     #Trwa_Krok_5;
      S     "Blok_Bledow_Program".Blad_Krok_5;
      A     #H_Blad;
      A     #Trwa_Krok_6;
      S     "Blok_Bledow_Program".Blad_Krok_6;
//Resetowanie bledu cyklu
      AN    #H_Blad;
      R     "Blok_Bledow_Program".Blad_Krok_1;
      R     "Blok_Bledow_Program".Blad_Krok_2;
      R     "Blok_Bledow_Program".Blad_Krok_3;
      R     "Blok_Bledow_Program".Blad_Krok_4;
      R     "Blok_Bledow_Program".Blad_Krok_5;
      R     "Blok_Bledow_Program".Blad_Krok_6;
NETWORK
TITLE =
//Zezwolenie na prace bindownicy
//0st ok
      AN    #H_Blad;
      A     #i_Pozycja_Obr_0st;
      AN    #i_Pozycja_Bandy_Lewo;
      A     #i_Fotokomorki_Pokryte;
      =     #H_Pozycja_0_st_ok;
//90st ok
      A     #i_Pozycja_Obr_90st;
      AN    #H_Blad;
      A     #i_Fotokomorki_Pokryte;
      =     #H_Pozycja_90_st_ok;
//180st
      AN    #H_Blad;
      A     #i_Pozycja_Obr_180st;
      AN    #i_Pozycja_Bandy_Prawo;
      A     #i_Fotokomorki_Pokryte;
      =     #H_Pozycja_180_st_ok;
//270st
      AN    #H_Blad;
      A     #i_Pozycja_Obr_270st;
      A     #i_Fotokomorki_Pokryte;
      =     #H_Pozycja_270_st_ok;
//Zezwolenie na prace bindownicy
      O     #H_Pozycja_0_st_ok;
      O     #H_Pozycja_90_st_ok;
      O     #H_Pozycja_180_st_ok;
      O     #H_Pozycja_270_st_ok;
      A     #i_Marka_Bezpieczenstwa;
      =     #o_Bind_Zez_Na_Prace;
END_FUNCTION_BLOCK

FUNCTION_BLOCK "Wybranie_Wjazdu"	// FB 50
VERSION : 0.1
VAR_INPUT
  Zajetosc_1_Lini : BOOL ;
  Zajetosc_2_Lini : BOOL ;
  Zezwolenie_Do_1_Lini : BOOL ;
  Zezwolenie_Do_2_Lini : BOOL ;
  Zabierz_Od_1_Lini : BOOL ;
  Zabierz_Od_2_Lini : BOOL ;
  Silniki_Nie_Pracuja : BOOL ;
END_VAR
VAR_IN_OUT
  Blokada_Kierunku_1 : BOOL ;
  Blokada_Kierunku_2 : BOOL ;
  Blokada : BOOL ;
END_VAR
VAR
  Czas_Kontrolny : SFB 4;
END_VAR
VAR_TEMP
  Temp_Help_1 : BOOL ;
  Temp_Help_2 : BOOL ;
END_VAR
BEGIN
NETWORK
TITLE =
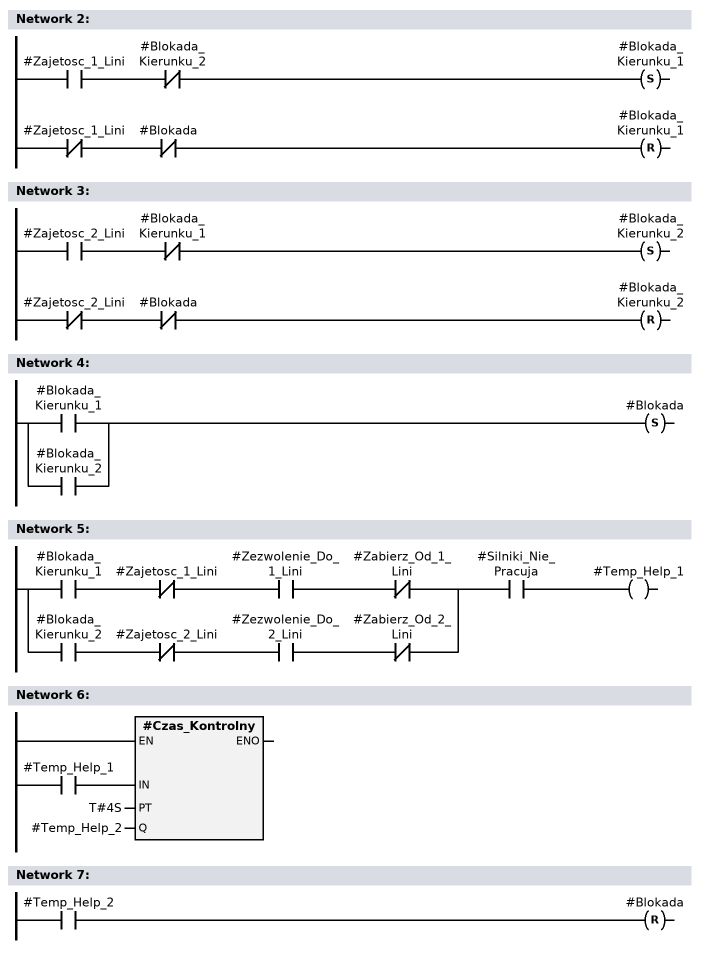
NETWORK
TITLE =
//Zarezerwowanie poboru palety z pierwszej lini
      A     #Zajetosc_1_Lini;
      AN    #Blokada_Kierunku_2;
      S     #Blokada_Kierunku_1;
      AN    #Zajetosc_1_Lini;
      AN    #Blokada;
      R     #Blokada_Kierunku_1;
      NOP   0;
NETWORK
TITLE =
//Zarezewowanie poboru palety z durgiej lini
      A     #Zajetosc_2_Lini;
      AN    #Blokada_Kierunku_1;
      S     #Blokada_Kierunku_2;
      AN    #Zajetosc_2_Lini;
      AN    #Blokada;
      R     #Blokada_Kierunku_2;
      NOP   0;
NETWORK
TITLE =
      A(;
      O     #Blokada_Kierunku_1;
      O     #Blokada_Kierunku_2;
      );
      S     #Blokada;
      NOP   0;
      NOP   0;
NETWORK
TITLE =
      A(;
      A     #Blokada_Kierunku_1;
      AN    #Zajetosc_1_Lini;
      A     #Zezwolenie_Do_1_Lini;
      AN    #Zabierz_Od_1_Lini;
      O;
      A     #Blokada_Kierunku_2;
      AN    #Zajetosc_2_Lini;
      A     #Zezwolenie_Do_2_Lini;
      AN    #Zabierz_Od_2_Lini;
      );
      A     #Silniki_Nie_Pracuja;
      =     #Temp_Help_1;
NETWORK
TITLE =
//Czas kontolny po ktorym nastepuje ponowne wybranie kierunku wjazdu
      A     #Temp_Help_1;
      =     L 1.0;
      BLD   103;
      CALL  #Czas_Kontrolny (
           IN                       := L 1.0,
           PT                       := T#4S,
           Q                        := #Temp_Help_2);
      NOP   0;
NETWORK
TITLE =
      A     #Temp_Help_2;
      R     #Blokada;
END_FUNCTION_BLOCK

FUNCTION_BLOCK "Obr_Na_Poz_1"	// FB 51
VERSION : 0.1
VAR_INPUT
  Jedz_Na_90st : BOOL ;
  Jedz_Na_0st : BOOL ;
  Czujnik_90st : BOOL ;
  Czujnik_0st : BOOL ;
  Czujnik_Ham_90st : BOOL ;
  Czujnik_Ham_0st : BOOL ;
  Odblowuj_Obrotnice : BOOL ;
END_VAR
VAR_OUTPUT
  Na_Pozycji_0st : BOOL ;	//Obrotnica na pozycji 0 stopni
  Na_Pozycji_90st : BOOL ;	//Obrotnica na pozycji 90 stopni
  Motor_Wolno : BOOL ;
  Odblokowanie_Rolek : BOOL ;
END_VAR
VAR_IN_OUT
  Talerz_w_Lewo : BOOL ;
  Talerz_w_Prawo : BOOL ;
END_VAR
VAR
  Czas_Dojscia : SFB 4;
  Czas_Startu : SFB 4;
  Help_Start : BOOL ;
END_VAR
VAR_TEMP
  Help_1 : BOOL ;
END_VAR
BEGIN
NETWORK
TITLE =
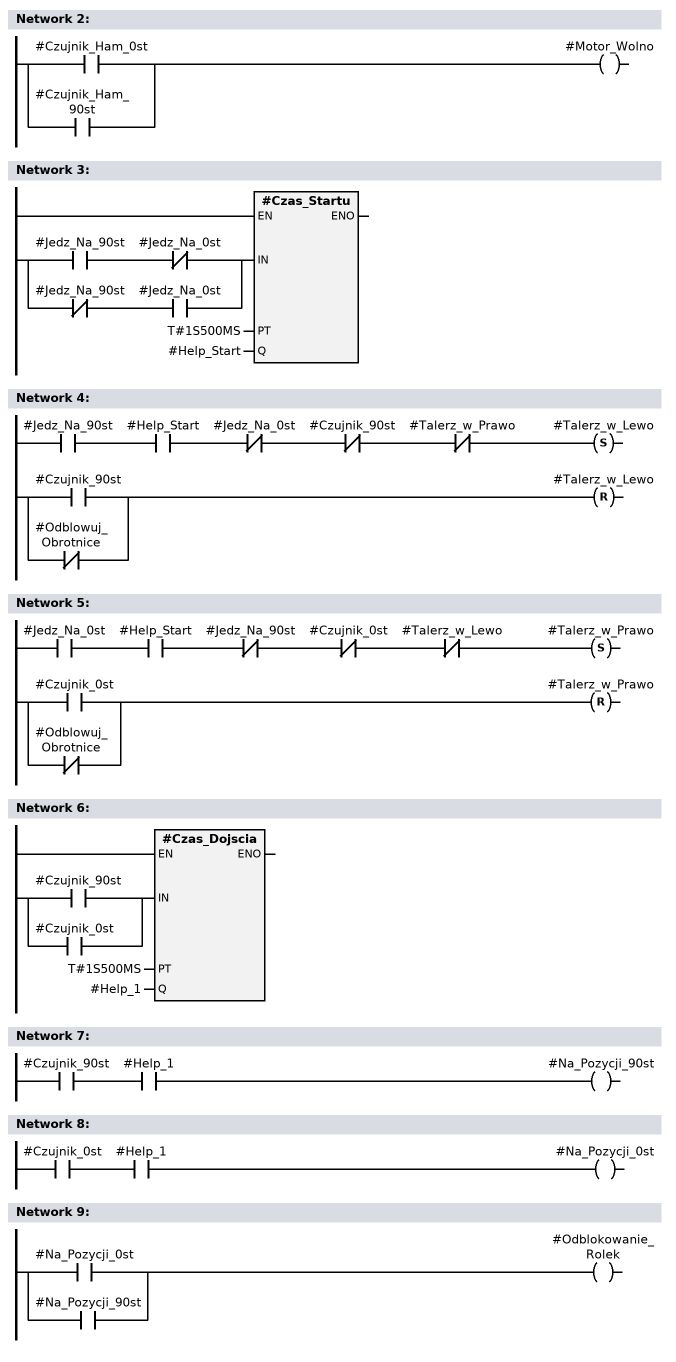
NETWORK
TITLE =
//Motor wolno gdy czujniki hamowania
      O     #Czujnik_Ham_0st;
      O     #Czujnik_Ham_90st;
      =     #Motor_Wolno;
NETWORK
TITLE =
      A(;
      A     #Jedz_Na_90st;
      AN    #Jedz_Na_0st;
      O;
      AN    #Jedz_Na_90st;
      A     #Jedz_Na_0st;
      );
      =     L 1.0;
      BLD   103;
      CALL  #Czas_Startu (
           IN                       := L 1.0,
           PT                       := T#1S500MS,
           Q                        := #Help_Start);
      NOP   0;
NETWORK
TITLE =
      A     #Jedz_Na_90st;
      A     #Help_Start;
      AN    #Jedz_Na_0st;
      AN    #Czujnik_90st;
      AN    #Talerz_w_Prawo;
      S     #Talerz_w_Lewo;
      A(;
      O     #Czujnik_90st;
      ON    #Odblowuj_Obrotnice;
      );
      R     #Talerz_w_Lewo;
      NOP   0;
NETWORK
TITLE =
      A     #Jedz_Na_0st;
      A     #Help_Start;
      AN    #Jedz_Na_90st;
      AN    #Czujnik_0st;
      AN    #Talerz_w_Lewo;
      S     #Talerz_w_Prawo;
      A(;
      O     #Czujnik_0st;
      ON    #Odblowuj_Obrotnice;
      );
      R     #Talerz_w_Prawo;
      NOP   0;
NETWORK
TITLE =
      A(;
      O     #Czujnik_90st;
      O     #Czujnik_0st;
      );
      =     L 1.0;
      BLD   103;
      CALL  #Czas_Dojscia (
           IN                       := L 1.0,
           PT                       := T#1S500MS,
           Q                        := #Help_1);
      NOP   0;
NETWORK
TITLE =
      A     #Czujnik_90st;
      A     #Help_1;
      =     #Na_Pozycji_90st;
NETWORK
TITLE =
      A     #Czujnik_0st;
      A     #Help_1;
      =     #Na_Pozycji_0st;
NETWORK
TITLE =
//Odblokowanie napedu rolkowego
      O     #Na_Pozycji_0st;
      O     #Na_Pozycji_90st;
      =     #Odblokowanie_Rolek;
END_FUNCTION_BLOCK

FUNCTION_BLOCK "Obr_Na_Poz_2"	// FB 52
//Funkcja sterujaca banda obrotowa. Programowana na jazde do roznych celow
VERSION : 0.1
VAR_INPUT
  Jedz_Na_90st : BOOL ;
  Jedz_Na_0st : BOOL ;
  Jedz_Na_45_st : BOOL ;
  Czujnik_90st : BOOL ;
  Czujnik_0st : BOOL ;
  Czujnik_45st_1 : BOOL ;
  Czujnik_45st_2 : BOOL ;
  Czujnik_Ham_90st : BOOL ;
  Czujnik_Ham_0st : BOOL ;
  Odblowuj_Obrotnice : BOOL ;
  Silownik_Bezpiecczny : BOOL ;
END_VAR
VAR_OUTPUT
  Na_Pozycji_0st : BOOL ;	//Obrotnica na pozycji 0 stopni
  Na_Pozycji_90st : BOOL ;	//Obrotnica na pozycji 90 stopni
  Na_Pozycji_45_st : BOOL ;
  Motor_Wolno : BOOL ;
  Odblokowanie_Rolek : BOOL ;
END_VAR
VAR_IN_OUT
  Talerz_w_Lewo : BOOL ;
  Talerz_w_Prawo : BOOL ;
END_VAR
VAR
  Czas_Dojscia : SFB 4;
  Czas_Startu : SFB 4;
  Help_Start : BOOL ;
END_VAR
VAR_TEMP
  Help_1 : BOOL ;
END_VAR
BEGIN
NETWORK
TITLE =
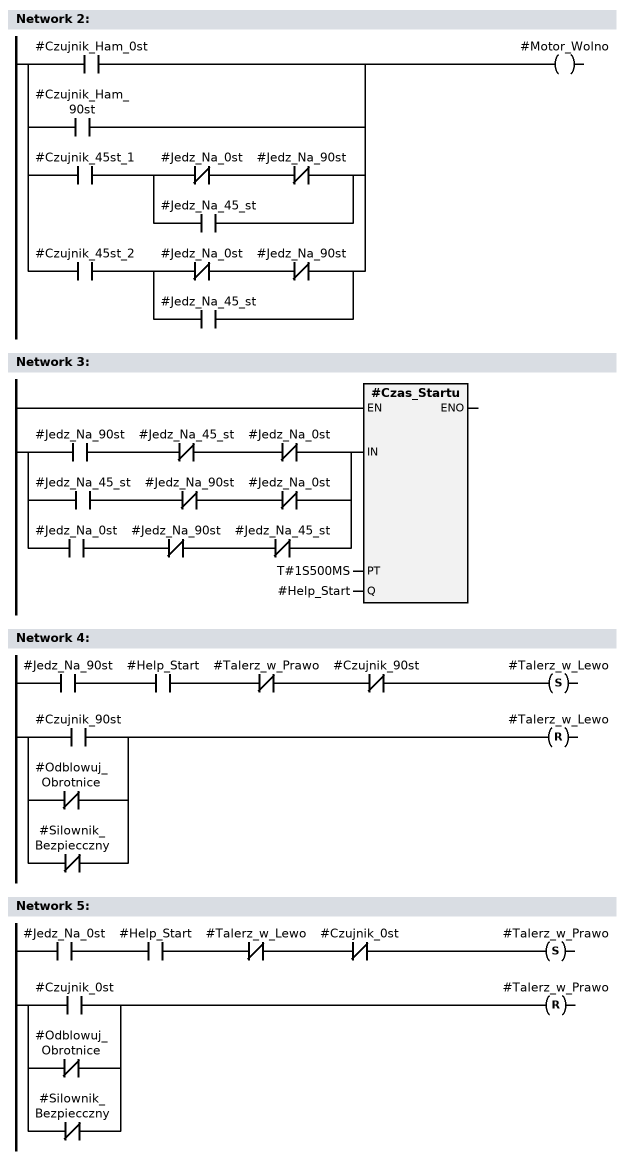
NETWORK
TITLE =
//Motor wolno gdy czujniki hamowania
      O     #Czujnik_Ham_0st;
      O     #Czujnik_Ham_90st;
      O;
      A     #Czujnik_45st_1;
      A(;
      AN    #Jedz_Na_0st;
      AN    #Jedz_Na_90st;
      O     #Jedz_Na_45_st;
      );
      O;
      A     #Czujnik_45st_2;
      A(;
      AN    #Jedz_Na_0st;
      AN    #Jedz_Na_90st;
      O     #Jedz_Na_45_st;
      );
      =     #Motor_Wolno;
NETWORK
TITLE =
      A(;
      A     #Jedz_Na_90st;
      AN    #Jedz_Na_45_st;
      AN    #Jedz_Na_0st;
      O;
      A     #Jedz_Na_45_st;
      AN    #Jedz_Na_90st;
      AN    #Jedz_Na_0st;
      O;
      A     #Jedz_Na_0st;
      AN    #Jedz_Na_90st;
      AN    #Jedz_Na_45_st;
      );
      =     L 1.0;
      BLD   103;
      CALL  #Czas_Startu (
           IN                       := L 1.0,
           PT                       := T#1S500MS,
           Q                        := #Help_Start);
      NOP   0;
NETWORK
TITLE =
      A     #Jedz_Na_90st;
      A     #Help_Start;
      AN    #Talerz_w_Prawo;
      AN    #Czujnik_90st;
      S     #Talerz_w_Lewo;
      A(;
      O     #Czujnik_90st;
      ON    #Odblowuj_Obrotnice;
      ON    #Silownik_Bezpiecczny;
      );
      R     #Talerz_w_Lewo;
      NOP   0;
NETWORK
TITLE =
      A     #Jedz_Na_0st;
      A     #Help_Start;
      AN    #Talerz_w_Lewo;
      AN    #Czujnik_0st;
      S     #Talerz_w_Prawo;
      A(;
      O     #Czujnik_0st;
      ON    #Odblowuj_Obrotnice;
      ON    #Silownik_Bezpiecczny;
      );
      R     #Talerz_w_Prawo;
      NOP   0;
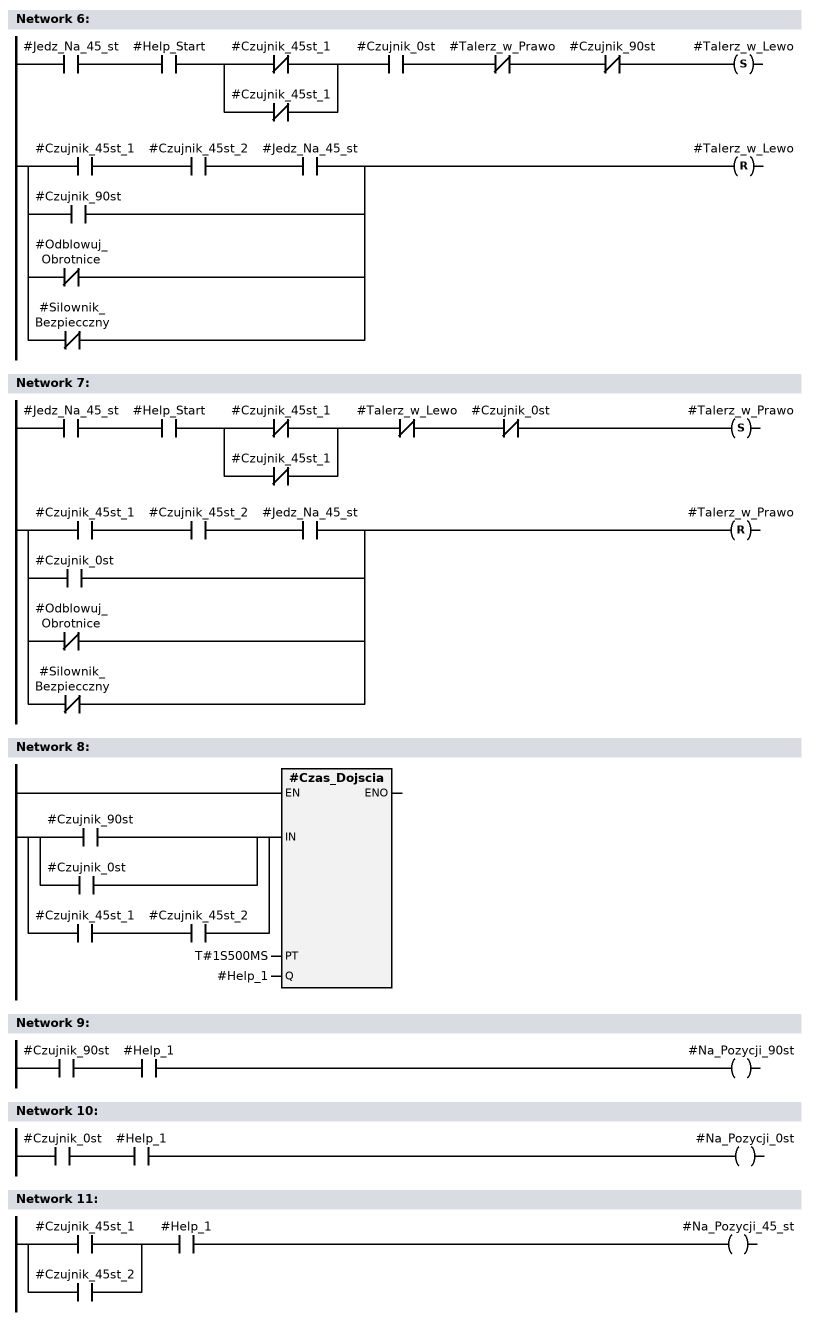
NETWORK
TITLE =
//Jazda na punkt 45st
      A     #Jedz_Na_45_st;
      A     #Help_Start;
      A(;
      ON    #Czujnik_45st_1;
      ON    #Czujnik_45st_1;
      );
      A     #Czujnik_0st;
      AN    #Talerz_w_Prawo;
      AN    #Czujnik_90st;
      S     #Talerz_w_Lewo;
      A(;
      A     #Czujnik_45st_1;
      A     #Czujnik_45st_2;
      A     #Jedz_Na_45_st;
      O     #Czujnik_90st;
      ON    #Odblowuj_Obrotnice;
      ON    #Silownik_Bezpiecczny;
      );
      R     #Talerz_w_Lewo;
      NOP   0;
NETWORK
TITLE =
//celowo brak czujnika 90st w ladzie
      A     #Jedz_Na_45_st;
      A     #Help_Start;
      A(;
      ON    #Czujnik_45st_1;
      ON    #Czujnik_45st_1;
      );
      AN    #Talerz_w_Lewo;
      AN    #Czujnik_0st;
      S     #Talerz_w_Prawo;
      A(;
      A     #Czujnik_45st_1;
      A     #Czujnik_45st_2;
      A     #Jedz_Na_45_st;
      O     #Czujnik_0st;
      ON    #Odblowuj_Obrotnice;
      ON    #Silownik_Bezpiecczny;
      );
      R     #Talerz_w_Prawo;
      NOP   0;
NETWORK
TITLE =
//Opoznienie przyjcia informacji o dojezdzie na pozycje
      A(;
      O     #Czujnik_90st;
      O     #Czujnik_0st;
      O;
      A     #Czujnik_45st_1;
      A     #Czujnik_45st_2;
      );
      =     L 1.0;
      BLD   103;
      CALL  #Czas_Dojscia (
           IN                       := L 1.0,
           PT                       := T#1S500MS,
           Q                        := #Help_1);
      NOP   0;
NETWORK
TITLE =
      A     #Czujnik_90st;
      A     #Help_1;
      =     #Na_Pozycji_90st;
NETWORK
TITLE =
      A     #Czujnik_0st;
      A     #Help_1;
      =     #Na_Pozycji_0st;
NETWORK
TITLE =
      A(;
      O     #Czujnik_45st_1;
      O     #Czujnik_45st_2;
      );
      A     #Help_1;
      =     #Na_Pozycji_45_st;
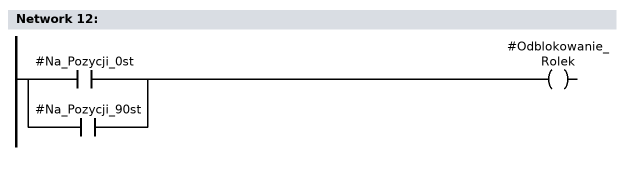
NETWORK
TITLE =
//Odblokowanie napedu rolkowego
      O     #Na_Pozycji_0st;
      O     #Na_Pozycji_90st;
      =     #Odblokowanie_Rolek;
END_FUNCTION_BLOCK

FUNCTION_BLOCK "Obr_Na_Poz_4"	// FB 54
//Funkcja sterujaca banda obrotowa. Programowana na jazde do roznych celow. 
//Zachowuje ona mo¿liwoœæ jazdy na 4 pozycje w zale¿noœci od po³o¿enia 
//inicjatorów 
//Kieunek jest wybierany ze wzgledu na wartosc liczbowa przyporzadkowana do 
//czujnikow. 
//
//0st_1- 1 czunik ostateczny oraz czujnik pozycji 0 stopni
//0st_2- 2 czujnik hamowania
//90st_1- 89 czujnik hamowania
//90st_2- 90 czujnik pozycji 90 stopni
//180st_1-179 czujnik hamowania 
//180st_2-180 czujnil pozycji 180 stopni
//270st_1-269 czujnik hamowania 
//270st_2-270 czujnik ostateczny oraz czujnik pozycji 270 stopni
//
//Czujniki ustawiane sa tak by przy obrocie we wlasciwym kierunku pracy najpierw 
//atakowany by³ czujnik hamowania a nastepnie czujnik pozycji docelowej
//Wyjatiem jest czujnik 0st(bo element startowy).
//
VERSION : 0.1
VAR_INPUT
  i_Marka_Bezpieczenstwa : BOOL ;
  i_Auto_Reczny : BOOL ;	//Auto-1,Reczny-0
  Zawsze_True : BOOL ;
  Jedz_Na_0st : BOOL ;
  Jedz_Na_90st : BOOL ;
  Jedz_Na_180st : BOOL ;
  Jedz_Na_270_st : BOOL ;
  Czujnik_0st_1 : BOOL ;
  Czujnik_0st_2 : BOOL ;
  Czujnik_90st_1 : BOOL ;
  Czujnik_90st_2 : BOOL ;
  Czujnik_180st_1 : BOOL ;
  Czujnik_180st_2 : BOOL ;
  Czujnik_270st_1 : BOOL ;
  Czujnik_270st_2 : BOOL ;
  Przycisk_Lewo : BOOL ;
  Przycisk_Prawo : BOOL ;
  s_Zez_Na_Obr : BOOL ;
  s_Ramie_Bind_w_Tyle : BOOL ;
END_VAR
VAR_OUTPUT
  Na_Pozycji_0st : BOOL ;	//Obrotnica na pozycji 0 stopni
  Na_Pozycji_90st : BOOL ;	//Obrotnica na pozycji 90 stopni
  Na_Pozycji_180st : BOOL ;
  Na_Pozycji_270st : BOOL ;
  Poz_Osiagnieta : BOOL ;	//Pozycja zadana osiagnieta
  s_Zez_Na_Rolki : BOOL ;	//Rolki odblowkowne je¿eli bindownica w poziomie do lini
  Motor_Wolno : BOOL ;
END_VAR
VAR_IN_OUT
  Talerz_w_Lewo : BOOL ;
  Talerz_w_Prawo : BOOL ;
  Pozycja : INT ;
END_VAR
VAR
  Czas_Dojscia : SFB 4;
  Czas_Startu : SFB 4;
  Help_Start : BOOL ;
  Help_Poz_0st : BOOL ;
  Help_Poz_90st : BOOL ;
  Help_Poz_180st : BOOL ;
  Help_Poz_270st : BOOL ;
  Help_A_Talerz_w_Prawo : BOOL ;	//CW
  Help_A_Talerz_w_Lewo : BOOL ;	//CCW
  Help_A_Motor_Wolno : BOOL ;
  Help_H_Talerz_w_Prawo : BOOL ;	//CW
  Help_H_Talerz_w_Lewo : BOOL ;	//CCW
  Help_H_Motor_Wolno : BOOL ;
  Help_Zbocze_0 : BOOL ;
  Help_Zbocze_1 : BOOL ;
  Help_Zbocze_2 : BOOL ;
  Help_Zbocze_3 : BOOL ;
  Help_Zbocze_4 : BOOL ;
  Silniki_nie_pracuja : BOOL ;
  Help_Opoznienie : BOOL ;
  Stop_Czas : BOOL ;
  help_18 : BOOL ;
  help_19 : BOOL ;
  help_20 : BOOL ;
END_VAR
VAR_TEMP
  Help_1 : BOOL ;
END_VAR
BEGIN
NETWORK
TITLE =
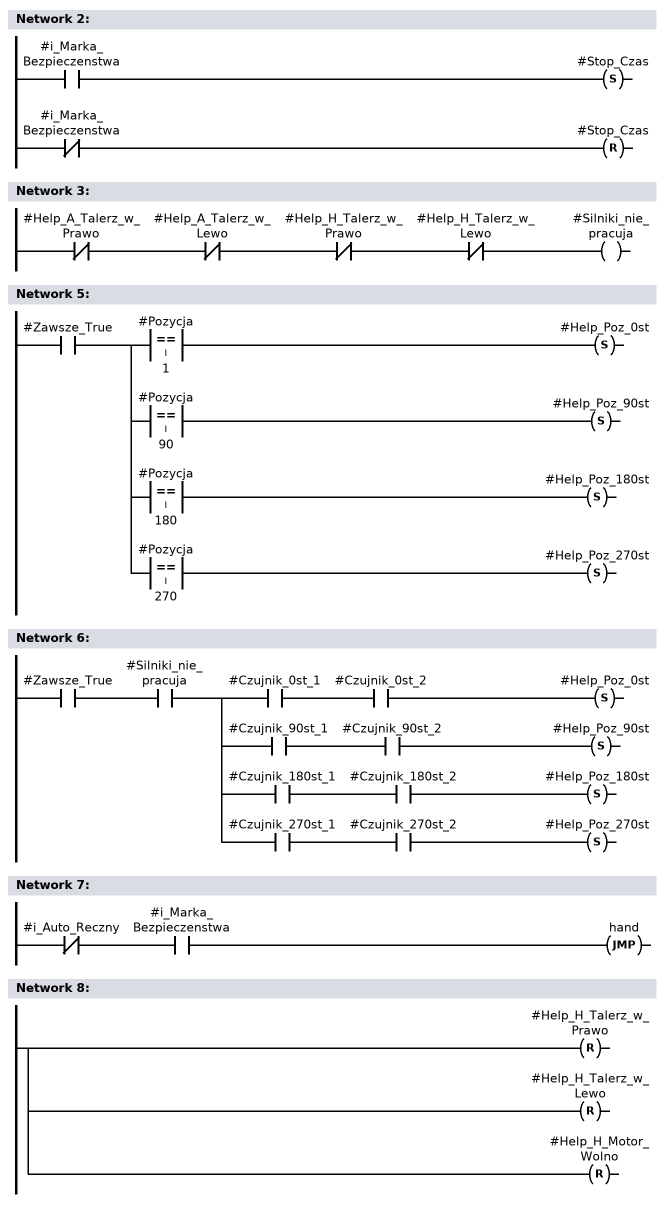
NETWORK
TITLE =
//ten network celowo jest wolny 
      A     #i_Marka_Bezpieczenstwa;
      S     #Stop_Czas;
      AN    #i_Marka_Bezpieczenstwa;
      R     #Stop_Czas;
NETWORK
TITLE =
//Sprawdzenie czy silniki nie pracuja 
      AN    #Help_A_Talerz_w_Prawo;
      AN    #Help_A_Talerz_w_Lewo;
      AN    #Help_H_Talerz_w_Prawo;
      AN    #Help_H_Talerz_w_Lewo;
      =     #Silniki_nie_pracuja;
NETWORK
TITLE =
      L     #Pozycja;
//********pozycja 0 stopni
//Pozycj 0 stopni obrotnica w pozycji wjazdu
      A     #Czujnik_0st_1;
      JCN   et_1;
      L     1;
      JU    poz;
et_1: NOP   0;
//zalaczony czujnik hamowania  samodzielnie
      A     #Czujnik_0st_2;
      AN    #Czujnik_0st_1;
      JCN   et_2;
      L     2;
      JU    poz;
et_2: NOP   0;
//********pozycja 90 stopni
//w kierunku cw najazd normalny z hamowaniem 
//w kierunku ccw najzd z minieciem pozycji + powrot
//czujnik 90 stopni hamowanie / w prawo
      O     #Help_A_Talerz_w_Prawo;
      O     #Help_H_Talerz_w_Prawo;
      A     #Czujnik_90st_1;
      AN    #Czujnik_90st_2;
      JCN   et_3;
      L     89;
      JU    poz;
et_3: NOP   0;
//czujnik 90 stopni pozycja  / w prawo
      O     #Help_A_Talerz_w_Prawo;
      O     #Help_H_Talerz_w_Prawo;
      A     #Czujnik_90st_2;
      JCN   et_4;
      L     90;
      JU    poz;
et_4: NOP   0;
//czujnik 90 stopni / w lewo
      O     #Help_A_Talerz_w_Lewo;
      O     #Help_H_Talerz_w_Lewo;
      A     #Czujnik_90st_2;
      JCN   e_13;
      L     91;
      JU    poz;
e_13: NOP   0;
//czujnik hamowania 90 stopni w lewo 
      O     #Help_A_Talerz_w_Lewo;
      O     #Help_H_Talerz_w_Lewo;
      A     #Czujnik_90st_1;
      AN    #Czujnik_90st_2;
      JCN   e_14;
      L     88;
      JU    poz;
e_14: NOP   0;
//********pozycja 180 stopni
//w kierunku ccw najzd z minieciem pozycji + powrot
//czujnik 180 stopni hamowanie
      O     #Help_A_Talerz_w_Prawo;
      O     #Help_H_Talerz_w_Prawo;
      A     #Czujnik_180st_1;
      AN    #Czujnik_180st_2;
      JCN   et_6;
      L     179;
      JU    poz;
et_6: NOP   0;
//czujnik 180 stopni pozycja
      O     #Help_A_Talerz_w_Prawo;
      O     #Help_H_Talerz_w_Prawo;
      A     #Czujnik_180st_2;
      JCN   et_7;
      L     180;
      JU    poz;
et_7: NOP   0;
//czujnik 180 stopni / w lewo
      O     #Help_A_Talerz_w_Lewo;
      O     #Help_H_Talerz_w_Lewo;
      A     #Czujnik_180st_2;
      JCN   e_16;
      L     181;
      JU    poz;
e_16: NOP   0;
//czujnik hamowania 180stopni w lewo 
      O     #Help_A_Talerz_w_Lewo;
      O     #Help_H_Talerz_w_Lewo;
      A     #Czujnik_180st_1;
      AN    #Czujnik_180st_2;
      JCN   e_17;
      L     178;
      JU    poz;
e_17: NOP   0;
//********pozycja 270 stopni
//270 stopni pozycja hamowania
      A     #Czujnik_270st_1;
      AN    #Czujnik_270st_2;
      JCN   et_8;
      L     269;
      JU    poz;
et_8: NOP   0;
//czujnik 270 stopni pozycja
      A     #Czujnik_270st_2;
      JCN   et_9;
      L     270;
      JU    poz;
et_9: NOP   0;
//Przypisanie wartosci pozycji
poz:  NOP   0;
      T     #Pozycja;
//sprawdz czy wartosci mieszcza sie w zakresie
      O(;
      L     #Pozycja;
      L     1;
      <I;
      );
      O(;
      L     #Pozycja;
      L     270;
      >I;
      );
      JCN   cv;
      L     100;
      T     #Pozycja;
cv:   NOP   0;
NETWORK
TITLE =
//Sprawdzenie pozycji dla recznego
      A     #Zawsze_True;
      =     L 1.0;
      A     L 1.0;
      A(;
      L     #Pozycja;
      L     1;
      ==I;
      );
      S     #Help_Poz_0st;
      A     L 1.0;
      A(;
      L     #Pozycja;
      L     90;
      ==I;
      );
      S     #Help_Poz_90st;
      A     L 1.0;
      A(;
      L     #Pozycja;
      L     180;
      ==I;
      );
      S     #Help_Poz_180st;
      A     L 1.0;
      A(;
      L     #Pozycja;
      L     270;
      ==I;
      );
      S     #Help_Poz_270st;
NETWORK
TITLE =
////Warunkowe przypisanie pozycji po glebszym bledzie
      A     #Zawsze_True;
      A     #Silniki_nie_pracuja;
      =     L 1.0;
      A     L 1.0;
      A     #Czujnik_0st_1;
      A     #Czujnik_0st_2;
      S     #Help_Poz_0st;
      A     L 1.0;
      A     #Czujnik_90st_1;
      A     #Czujnik_90st_2;
      S     #Help_Poz_90st;
      A     L 1.0;
      A     #Czujnik_180st_1;
      A     #Czujnik_180st_2;
      S     #Help_Poz_180st;
      A     L 1.0;
      A     #Czujnik_270st_1;
      A     #Czujnik_270st_2;
      S     #Help_Poz_270st;
NETWORK
TITLE =
//jazda na pozycje zadana
//skocz jezeli tryb reczny
      AN    #i_Auto_Reczny;
      A     #i_Marka_Bezpieczenstwa;
      JC    hand;
NETWORK
TITLE =
//Kasowanie bitow z trybu recznego 
      SET;
      R     #Help_H_Talerz_w_Prawo;
      R     #Help_H_Talerz_w_Lewo;
      R     #Help_H_Motor_Wolno;
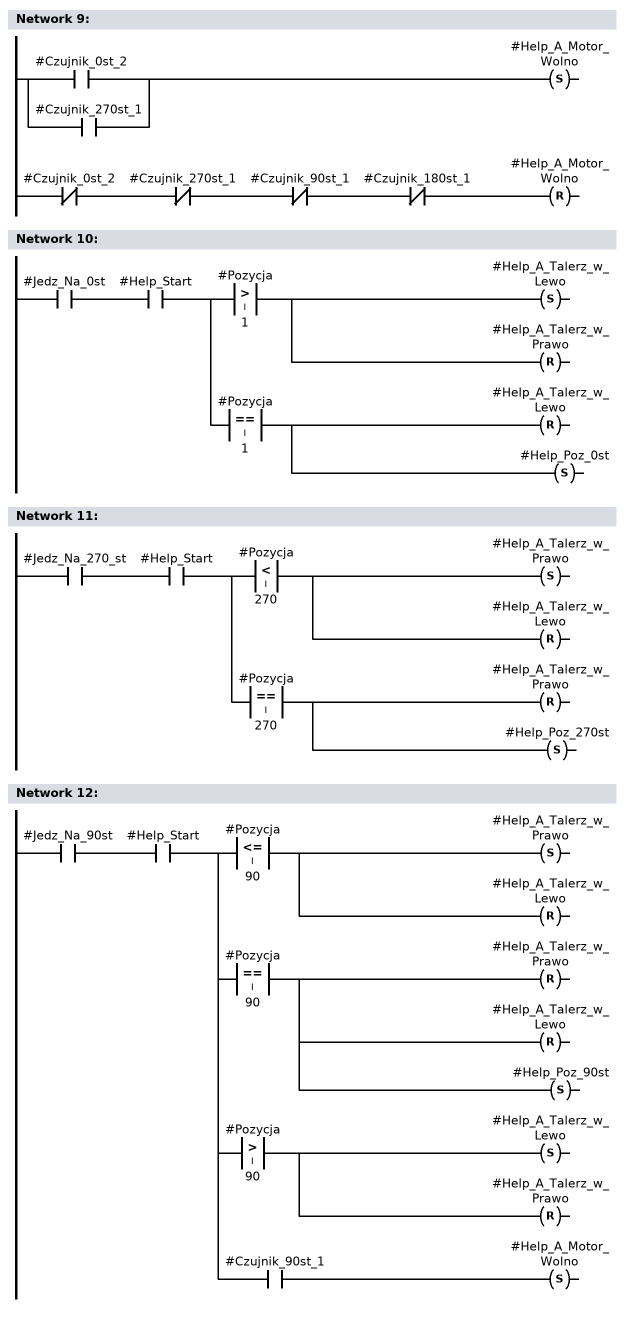
NETWORK
TITLE =
//Zalaczenie trybu wolnego. Wylaczony gdy zaden z czujnikow nie jest zalaczony
      A(;
      O     #Czujnik_0st_2;
      O     #Czujnik_270st_1;
      );
      S     #Help_A_Motor_Wolno;
      AN    #Czujnik_0st_2;
      AN    #Czujnik_270st_1;
      AN    #Czujnik_90st_1;
      AN    #Czujnik_180st_1;
      R     #Help_A_Motor_Wolno;
      NOP   0;
NETWORK
TITLE =
//Jazda na pozycje 0 st
//
      A     #Jedz_Na_0st;
      A     #Help_Start;
      =     L 1.0;
      A     L 1.0;
      A(;
      L     #Pozycja;
      L     1;
      >I;
      );
      S     #Help_A_Talerz_w_Lewo;
      R     #Help_A_Talerz_w_Prawo;
      A     L 1.0;
      A(;
      L     #Pozycja;
      L     1;
      ==I;
      );
      R     #Help_A_Talerz_w_Lewo;
      S     #Help_Poz_0st;
NETWORK
TITLE =
//Jazda na pozycje 270st 
//
      A     #Jedz_Na_270_st;
      A     #Help_Start;
      =     L 1.0;
      A     L 1.0;
      A(;
      L     #Pozycja;
      L     270;
      <I;
      );
      S     #Help_A_Talerz_w_Prawo;
      R     #Help_A_Talerz_w_Lewo;
      A     L 1.0;
      A(;
      L     #Pozycja;
      L     270;
      ==I;
      );
      R     #Help_A_Talerz_w_Prawo;
      S     #Help_Poz_270st;
NETWORK
TITLE =
//Jazda na 90 st od strony lewej i od strony prawej. Gdy najazd od strony lewej 
//najpierw jest hamowanie talerza nastepnie zatrzymanie. Gdy najazd od strony 
//prawej nastepuje miniecie czujnika nastepnie zatrzymanie i cofniecie
//
//
      A     #Jedz_Na_90st;
      A     #Help_Start;
      =     L 1.0;
      A     L 1.0;
      A(;
      L     #Pozycja;
      L     90;
      <=I;
      );
      S     #Help_A_Talerz_w_Prawo;
      R     #Help_A_Talerz_w_Lewo;
      A     L 1.0;
      A(;
      L     #Pozycja;
      L     90;
      ==I;
      );
      R     #Help_A_Talerz_w_Prawo;
      R     #Help_A_Talerz_w_Lewo;
      S     #Help_Poz_90st;
      A     L 1.0;
      A(;
      L     #Pozycja;
      L     90;
      >I;
      );
      S     #Help_A_Talerz_w_Lewo;
      R     #Help_A_Talerz_w_Prawo;
      A     L 1.0;
      A     #Czujnik_90st_1;
      S     #Help_A_Motor_Wolno;
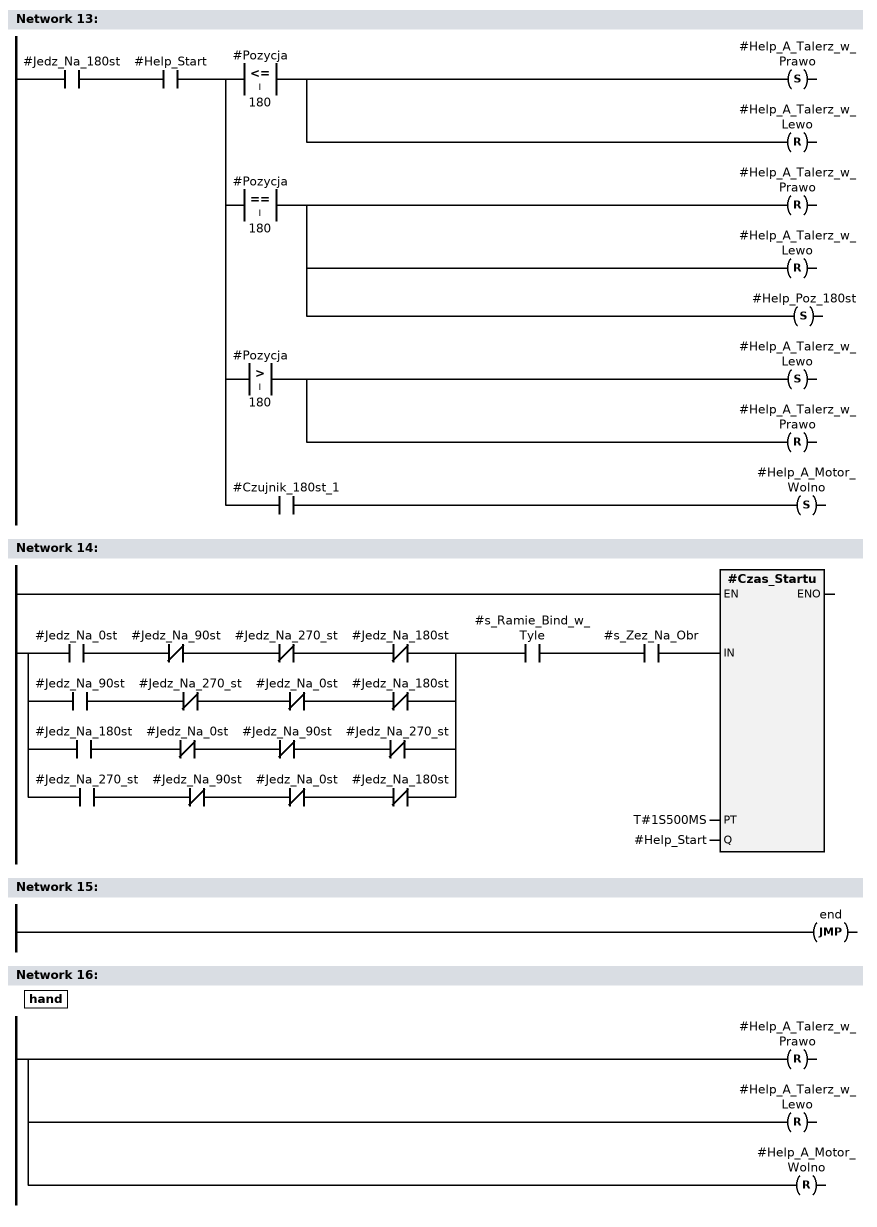
NETWORK
TITLE =
//Jazda na 180 st od strony lewej i od strony prawej. Gdy najazd od strony lewej 
//najpierw jest hamowanie talerza nastepnie zatrzymanie. Gdy najazd od strony 
//prawej nastepuje miniecie czujnika nastepnie zatrzymanie i cofniecie
//
//
      A     #Jedz_Na_180st;
      A     #Help_Start;
      =     L 1.0;
      A     L 1.0;
      A(;
      L     #Pozycja;
      L     180;
      <=I;
      );
      S     #Help_A_Talerz_w_Prawo;
      R     #Help_A_Talerz_w_Lewo;
      A     L 1.0;
      A(;
      L     #Pozycja;
      L     180;
      ==I;
      );
      R     #Help_A_Talerz_w_Prawo;
      R     #Help_A_Talerz_w_Lewo;
      S     #Help_Poz_180st;
      A     L 1.0;
      A(;
      L     #Pozycja;
      L     180;
      >I;
      );
      S     #Help_A_Talerz_w_Lewo;
      R     #Help_A_Talerz_w_Prawo;
      A     L 1.0;
      A     #Czujnik_180st_1;
      S     #Help_A_Motor_Wolno;
NETWORK
TITLE =
//Opoznienie startu po wydaniu rozkazu
      A(;
      A     #Jedz_Na_0st;
      AN    #Jedz_Na_90st;
      AN    #Jedz_Na_270_st;
      AN    #Jedz_Na_180st;
      O;
      A     #Jedz_Na_90st;
      AN    #Jedz_Na_270_st;
      AN    #Jedz_Na_0st;
      AN    #Jedz_Na_180st;
      O;
      A     #Jedz_Na_180st;
      AN    #Jedz_Na_0st;
      AN    #Jedz_Na_90st;
      AN    #Jedz_Na_270_st;
      O;
      A     #Jedz_Na_270_st;
      AN    #Jedz_Na_90st;
      AN    #Jedz_Na_0st;
      AN    #Jedz_Na_180st;
      );
      A     #s_Ramie_Bind_w_Tyle;
      A     #s_Zez_Na_Obr;
      =     L 1.0;
      BLD   103;
      CALL  #Czas_Startu (
           IN                       := L 1.0,
           PT                       := T#1S500MS,
           Q                        := #Help_Start);
      NOP   0;
NETWORK
TITLE =
//Koniec tryby automatycznego
//
      JU    end;
NETWORK
TITLE =
//tryb reczny
hand: NOP   0;
      SET;
      R     #Help_A_Talerz_w_Prawo;
      R     #Help_A_Talerz_w_Lewo;
      R     #Help_A_Motor_Wolno;
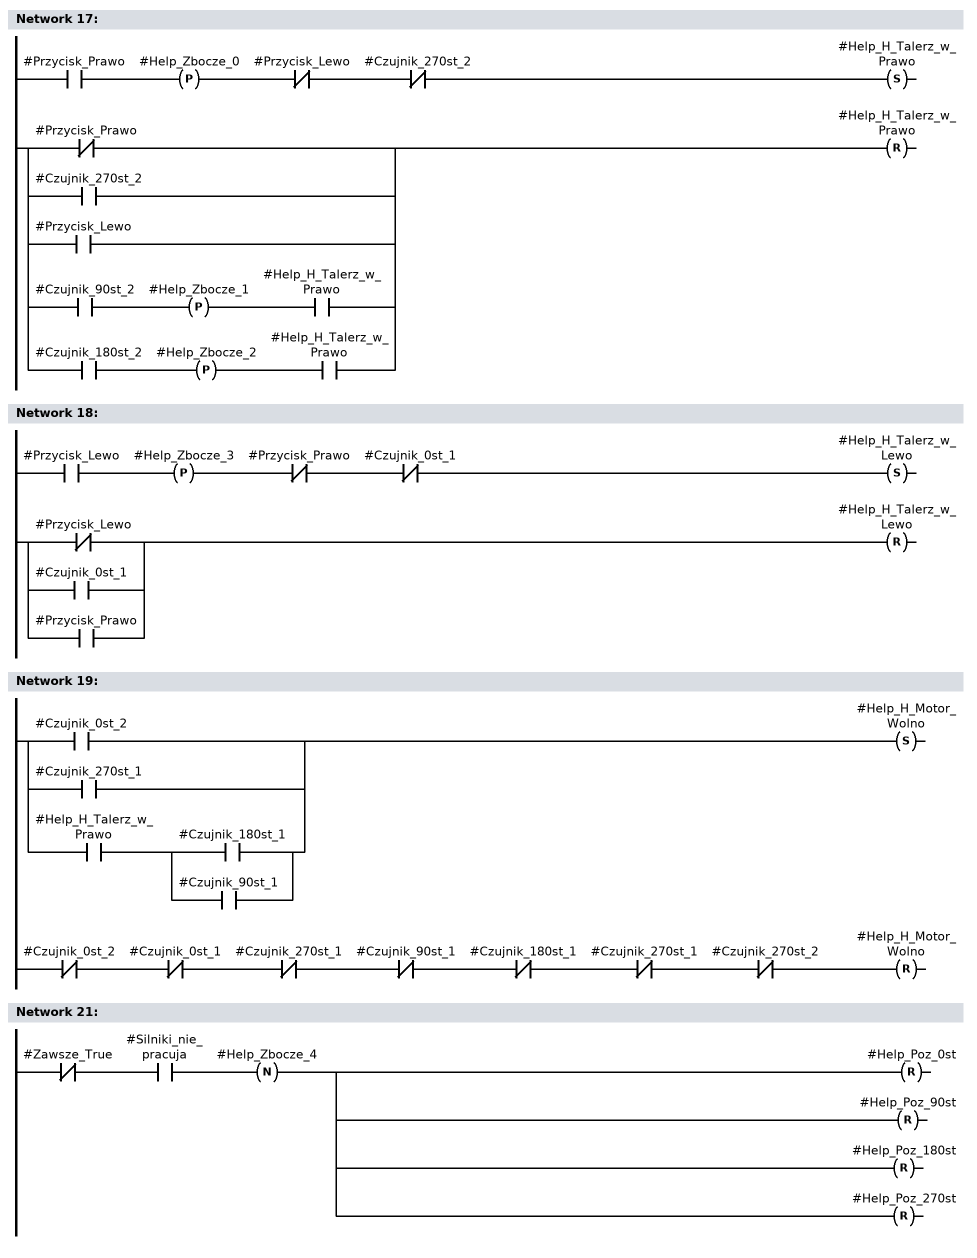
NETWORK
TITLE =
//Ruch talerza w prawo i zatrzymywanie sie na pozycji
//
      A     #Przycisk_Prawo;
      FP    #Help_Zbocze_0;
      AN    #Przycisk_Lewo;
      AN    #Czujnik_270st_2;
      S     #Help_H_Talerz_w_Prawo;
      A(;
      ON    #Przycisk_Prawo;
      O     #Czujnik_270st_2;
      O     #Przycisk_Lewo;
      O(;
      A     #Czujnik_90st_2;
      FP    #Help_Zbocze_1;
      A     #Help_H_Talerz_w_Prawo;
      );
      O(;
      A     #Czujnik_180st_2;
      FP    #Help_Zbocze_2;
      A     #Help_H_Talerz_w_Prawo;
      );
      );
      R     #Help_H_Talerz_w_Prawo;
      NOP   0;
NETWORK
TITLE =
//Ruch talerza w lewo. Zatrzymanie tylko na skrajnych pozycjach
//
      A     #Przycisk_Lewo;
      FP    #Help_Zbocze_3;
      AN    #Przycisk_Prawo;
      AN    #Czujnik_0st_1;
      S     #Help_H_Talerz_w_Lewo;
      A(;
      ON    #Przycisk_Lewo;
      O     #Czujnik_0st_1;
      O     #Przycisk_Prawo;
      );
      R     #Help_H_Talerz_w_Lewo;
      NOP   0;
NETWORK
TITLE =
//Zwolnienie predkosci gdy jazda w trybie recznym 
      A(;
      O     #Czujnik_0st_2;
      O     #Czujnik_270st_1;
      O;
      A     #Help_H_Talerz_w_Prawo;
      A(;
      O     #Czujnik_180st_1;
      O     #Czujnik_90st_1;
      );
      );
      S     #Help_H_Motor_Wolno;
      AN    #Czujnik_0st_2;
      AN    #Czujnik_0st_1;
      AN    #Czujnik_270st_1;
      AN    #Czujnik_90st_1;
      AN    #Czujnik_180st_1;
      AN    #Czujnik_270st_1;
      AN    #Czujnik_270st_2;
      R     #Help_H_Motor_Wolno;
      NOP   0;
NETWORK
TITLE =
end:  NOP   0;
NETWORK
TITLE =
//resetowanie pozycji gdy silniki rusza.
//Rozkaz kasowania wyciety
      AN    #Zawsze_True;
      A     #Silniki_nie_pracuja;
      FN    #Help_Zbocze_4;
      R     #Help_Poz_0st;
      R     #Help_Poz_90st;
      R     #Help_Poz_180st;
      R     #Help_Poz_270st;
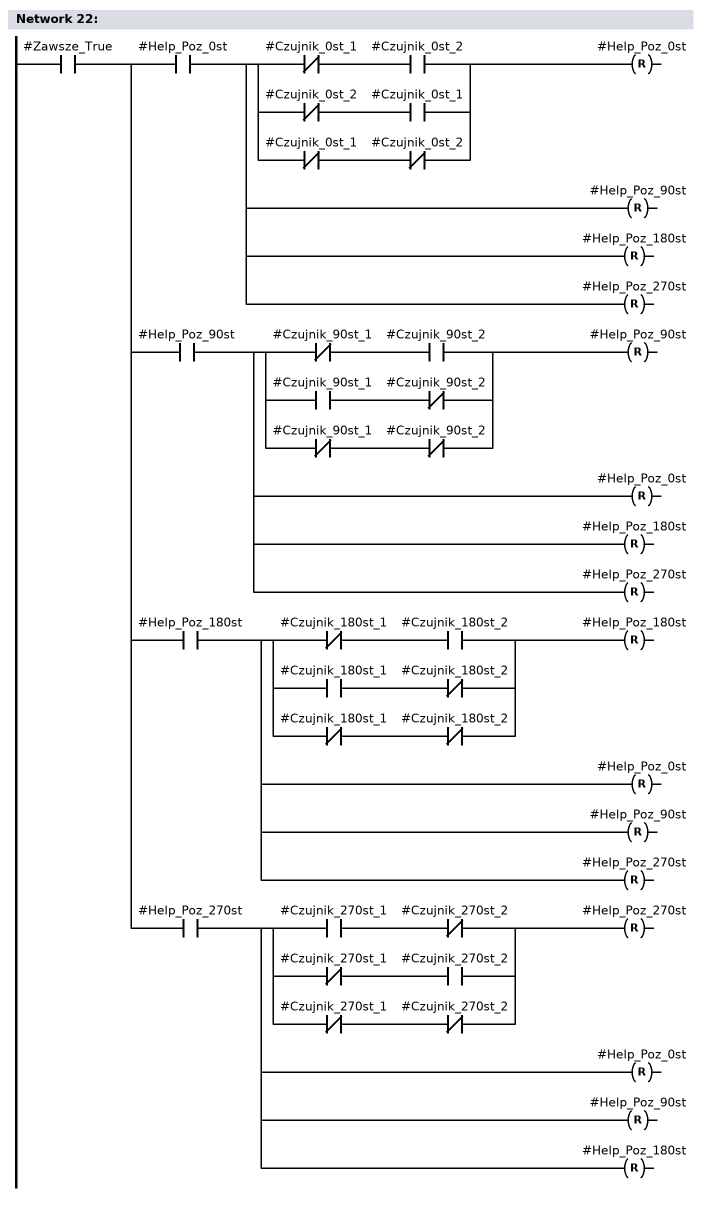
NETWORK
TITLE =
//The can be only one.
      A     #Zawsze_True;
      =     L 1.0;
      A     L 1.0;
      A     #Help_Poz_0st;
      =     L 1.1;
      A     L 1.1;
      A(;
      AN    #Czujnik_0st_1;
      A     #Czujnik_0st_2;
      O;
      AN    #Czujnik_0st_2;
      A     #Czujnik_0st_1;
      O;
      AN    #Czujnik_0st_1;
      AN    #Czujnik_0st_2;
      );
      R     #Help_Poz_0st;
      A     L 1.1;
      BLD   102;
      R     #Help_Poz_90st;
      A     L 1.1;
      BLD   102;
      R     #Help_Poz_180st;
      A     L 1.1;
      BLD   102;
      R     #Help_Poz_270st;
      A     L 1.0;
      A     #Help_Poz_90st;
      =     L 1.1;
      A     L 1.1;
      A(;
      AN    #Czujnik_90st_1;
      A     #Czujnik_90st_2;
      O;
      A     #Czujnik_90st_1;
      AN    #Czujnik_90st_2;
      O;
      AN    #Czujnik_90st_1;
      AN    #Czujnik_90st_2;
      );
      R     #Help_Poz_90st;
      A     L 1.1;
      BLD   102;
      R     #Help_Poz_0st;
      A     L 1.1;
      BLD   102;
      R     #Help_Poz_180st;
      A     L 1.1;
      BLD   102;
      R     #Help_Poz_270st;
      A     L 1.0;
      A     #Help_Poz_180st;
      =     L 1.1;
      A     L 1.1;
      A(;
      AN    #Czujnik_180st_1;
      A     #Czujnik_180st_2;
      O;
      A     #Czujnik_180st_1;
      AN    #Czujnik_180st_2;
      O;
      AN    #Czujnik_180st_1;
      AN    #Czujnik_180st_2;
      );
      R     #Help_Poz_180st;
      A     L 1.1;
      BLD   102;
      R     #Help_Poz_0st;
      A     L 1.1;
      BLD   102;
      R     #Help_Poz_90st;
      A     L 1.1;
      BLD   102;
      R     #Help_Poz_270st;
      A     L 1.0;
      A     #Help_Poz_270st;
      =     L 1.1;
      A     L 1.1;
      A(;
      A     #Czujnik_270st_1;
      AN    #Czujnik_270st_2;
      O;
      AN    #Czujnik_270st_1;
      A     #Czujnik_270st_2;
      O;
      AN    #Czujnik_270st_1;
      AN    #Czujnik_270st_2;
      );
      R     #Help_Poz_270st;
      A     L 1.1;
      BLD   102;
      R     #Help_Poz_0st;
      A     L 1.1;
      BLD   102;
      R     #Help_Poz_90st;
      A     L 1.1;
      BLD   102;
      R     #Help_Poz_180st;
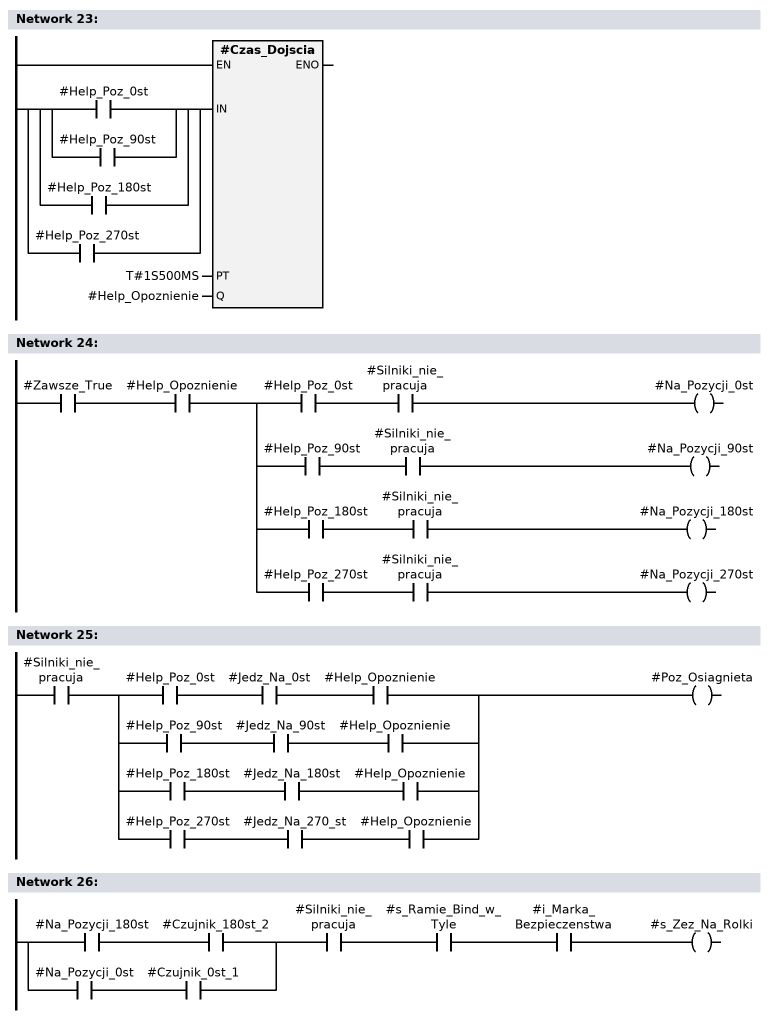
NETWORK
TITLE =
//Opoznienie potwierdzenia pozycji
      A(;
      O     #Help_Poz_0st;
      O     #Help_Poz_90st;
      O     #Help_Poz_180st;
      O     #Help_Poz_270st;
      );
      =     L 1.0;
      BLD   103;
      CALL  #Czas_Dojscia (
           IN                       := L 1.0,
           PT                       := T#1S500MS,
           Q                        := #Help_Opoznienie);
      NOP   0;
NETWORK
TITLE =
//przypisanie pozycji
//
      A     #Zawsze_True;
      A     #Help_Opoznienie;
      =     L 1.0;
      A     L 1.0;
      A     #Help_Poz_0st;
      A     #Silniki_nie_pracuja;
      =     #Na_Pozycji_0st;
      A     L 1.0;
      A     #Help_Poz_90st;
      A     #Silniki_nie_pracuja;
      =     #Na_Pozycji_90st;
      A     L 1.0;
      A     #Help_Poz_180st;
      A     #Silniki_nie_pracuja;
      =     #Na_Pozycji_180st;
      A     L 1.0;
      A     #Help_Poz_270st;
      A     #Silniki_nie_pracuja;
      =     #Na_Pozycji_270st;
NETWORK
TITLE =
//Potwierdzenie osiagniecia pozycji
      A     #Silniki_nie_pracuja;
      A(;
      A     #Help_Poz_0st;
      A     #Jedz_Na_0st;
      A     #Help_Opoznienie;
      O;
      A     #Help_Poz_90st;
      A     #Jedz_Na_90st;
      A     #Help_Opoznienie;
      O;
      A     #Help_Poz_180st;
      A     #Jedz_Na_180st;
      A     #Help_Opoznienie;
      O;
      A     #Help_Poz_270st;
      A     #Jedz_Na_270_st;
      A     #Help_Opoznienie;
      );
      =     #Poz_Osiagnieta;
NETWORK
TITLE =
//Warunek odblokowanch rolek
      A(;
      A     #Na_Pozycji_180st;
      A     #Czujnik_180st_2;
      O;
      A     #Na_Pozycji_0st;
      A     #Czujnik_0st_1;
      );
      A     #Silniki_nie_pracuja;
      A     #s_Ramie_Bind_w_Tyle;
      A     #i_Marka_Bezpieczenstwa;
      =     #s_Zez_Na_Rolki;
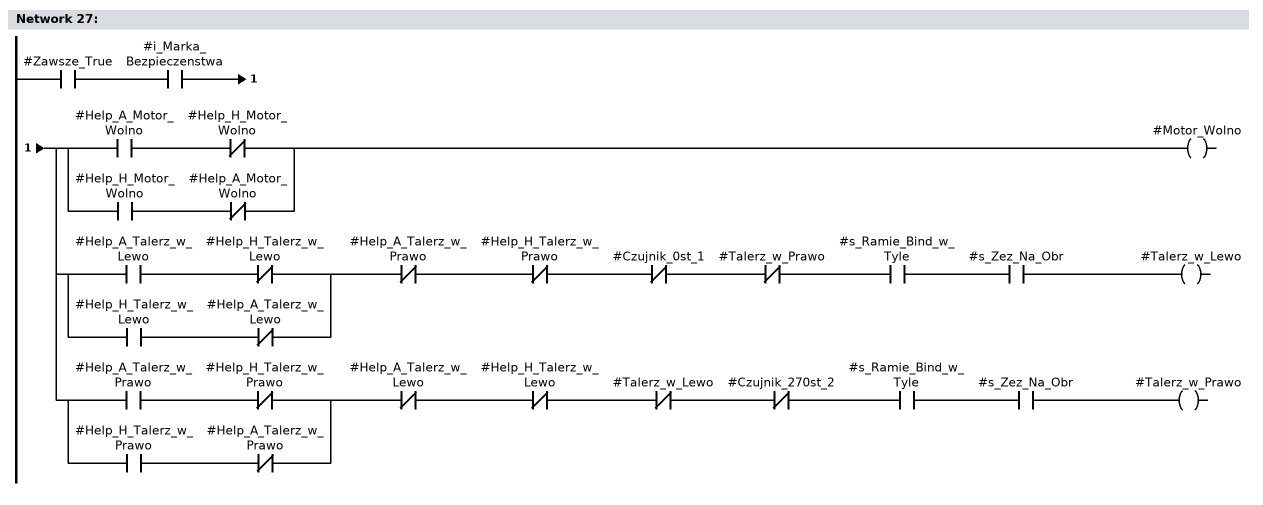
NETWORK
TITLE =
//wykonianie obrotu warunki jazdy
      A     #Zawsze_True;
      A     #i_Marka_Bezpieczenstwa;
      =     L 1.0;
      A     L 1.0;
      A(;
      A     #Help_A_Motor_Wolno;
      AN    #Help_H_Motor_Wolno;
      O;
      A     #Help_H_Motor_Wolno;
      AN    #Help_A_Motor_Wolno;
      );
      =     #Motor_Wolno;
      A     L 1.0;
      A(;
      A     #Help_A_Talerz_w_Lewo;
      AN    #Help_H_Talerz_w_Lewo;
      O;
      A     #Help_H_Talerz_w_Lewo;
      AN    #Help_A_Talerz_w_Lewo;
      );
      AN    #Help_A_Talerz_w_Prawo;
      AN    #Help_H_Talerz_w_Prawo;
      AN    #Czujnik_0st_1;
      AN    #Talerz_w_Prawo;
      A     #s_Ramie_Bind_w_Tyle;
      A     #s_Zez_Na_Obr;
      =     #Talerz_w_Lewo;
      A     L 1.0;
      A(;
      A     #Help_A_Talerz_w_Prawo;
      AN    #Help_H_Talerz_w_Prawo;
      O;
      A     #Help_H_Talerz_w_Prawo;
      AN    #Help_A_Talerz_w_Prawo;
      );
      AN    #Help_A_Talerz_w_Lewo;
      AN    #Help_H_Talerz_w_Lewo;
      AN    #Talerz_w_Lewo;
      AN    #Czujnik_270st_2;
      A     #s_Ramie_Bind_w_Tyle;
      A     #s_Zez_Na_Obr;
      =     #Talerz_w_Prawo;
END_FUNCTION_BLOCK

FUNCTION_BLOCK "Pozycjonowanie_Bandy"	// FB 55
//Funcja odpowiada za jazde rolek na pozycje zgodnie z rozkazem 
VERSION : 0.1
VAR_INPUT
  i_Auto_Reczny : BOOL ;
  Stop_Bezpieczenistwa : BOOL ;
  Pozycjonuj_Lewo : BOOL ;
  Pozycjonuj_Prawo : BOOL ;
  Powrot_Poz : BOOL ;
  Foto_Przod : BOOL ;
  Foto_Tyl : BOOL ;
  i_Zez_Na_Rolki : BOOL ;
  Reset : BOOL ;
  Czas_Prawo : TIME ;
  Czas_Lewo : TIME ;
  Czas_Kontrolny : TIME ;
  Czas_Pow_Prawo : TIME ;
  Czas_Pow_Lewo : TIME ;
  Blokada_Obrotu_1 : BOOL ;
  i_Resetuj_Srodek : BOOL ;	//Przesow rolek z innego trybu
END_VAR
VAR_OUTPUT
  Potw_Pozycji : BOOL ;
  Pozycja_Lewo : BOOL ;	//Odniesienie do 0st
  Pozycja_Prawo : BOOL ;	//Odniesienie do 0st
  Pozycja_Srodek : BOOL ;
  Motor_Lewo : BOOL ;
  Motor_Prawo : BOOL ;
  Motor_Wolno : BOOL ;
  Zez_Na_Obrot : BOOL ;
  Blad_Pozycjowania : BOOL ;
END_VAR
VAR
  Pozycja_Wyjsciowa : BOOL ;
  Tim_Jazdy_Prawo : FB 20;
  Tim_Jazdy_Lewo : FB 20;
  Tim_Kon_Prawo : FB 20;	//Timmer kontrolny prawo
  Tim_Kon_Lewo : FB 20;	//Timmer kontrolny lewo
  Help_Motor_Prawo : BOOL ;
  Help_Motor_Lewo : BOOL ;
  H_Repozycj_Prawo : BOOL ;
  H_Repozycj_Lewo : BOOL ;
  Help_Motor_Wolno : BOOL ;
  H_Powr_od_Prawo_1 : BOOL ;
  H_Powr_od_Lewo_1 : BOOL ;
  H_Powr_Prawo : BOOL ;
  H_Powr_Lewo : BOOL ;
  Help_Poz_Prawo : BOOL ;
  Help_Poz_Lewo : BOOL ;
  Pozycj_Warunkowe : BOOL ;
  Skrajne_Prawo : BOOL ;
  Skrajne_Lewo : BOOL ;
  Zbocze_1 : BOOL ;
  Zbocze_2 : BOOL ;
  H6 : BOOL ;
  H7 : BOOL ;
  H8 : BOOL ;
  H9 : BOOL ;
  H10 : BOOL ;
END_VAR
VAR_TEMP
  Temp_Help_1 : BOOL ;
  Temp_Help_2 : BOOL ;
  Temp_Help_3 : BOOL ;
  Czas_Aktualny : TIME ;
END_VAR
BEGIN
NETWORK
TITLE =
      A     #Foto_Przod;
      A     #Foto_Tyl;
      A     #Pozycja_Srodek;
      A     #i_Zez_Na_Rolki;	//rolki sa odblokowane w pozycji 0st lub 180st
      =     #Pozycja_Wyjsciowa;
      O     #Help_Motor_Lewo;
      O     #Help_Motor_Prawo;
      R     #Potw_Pozycji;
//warunkowe pozycjonowanie 
NETWORK
TITLE =
//Pozycjonowanie prawo
//Pozycjonowanie w prawo
      A     #i_Zez_Na_Rolki;
      A     #Pozycjonuj_Prawo;
      A     #Pozycja_Wyjsciowa;
      S     #Help_Motor_Prawo;
      S     #Help_Motor_Wolno;
      S     #Help_Poz_Prawo;
      R     #Pozycja_Srodek;
      CALL  #Tim_Jazdy_Prawo (
           IN                       := #Help_Poz_Prawo,
           STOP                     := #Stop_Bezpieczenistwa,
           PT                       := #Czas_Prawo,
           Q_0                      := #Temp_Help_2,
           ET                       := #Czas_Aktualny);
      A     #Temp_Help_2;
      O;
      A     #Help_Poz_Prawo;
      AN    #Foto_Przod;
      S     #Pozycja_Prawo;
      S     #Potw_Pozycji;
      R     #Help_Motor_Prawo;
      R     #Help_Motor_Wolno;
      R     #Help_Poz_Prawo;
//Powrot z pozycjonowania. 
//Zjazd z fotokomorki aby zrobic ponowny najazd
      O(;
      A     #Foto_Przod;
      A     #Pozycja_Prawo;
      A     #Powrot_Poz;
      AN    #H_Powr_od_Prawo_1;
      );
      O(;
      A     #Pozycj_Warunkowe;
      );
      S     #Help_Motor_Prawo;
      S     #Help_Motor_Wolno;
      S     #H_Repozycj_Prawo;
      R     #Pozycja_Prawo;
//koniec zjazdu z fotokomorki
      AN    #Foto_Przod;
      A     #H_Repozycj_Prawo;
      R     #Help_Motor_Prawo;
      R     #Help_Motor_Wolno;
      R     #H_Repozycj_Prawo;
      S     #Skrajne_Prawo;
//powrot na pozycje na srodku obrtnicy
      A(;
      O     #Powrot_Poz;
      O     #Skrajne_Prawo;
      O     #Pozycj_Warunkowe;
      );
      A(;
      O     #Pozycja_Prawo;
      O     #Skrajne_Prawo;
      );
      AN    #Foto_Przod;
      S     #Help_Motor_Lewo;
      S     #Help_Motor_Wolno;
      S     #H_Powr_od_Prawo_1;
      R     #Help_Motor_Prawo;
      R     #Pozycja_Prawo;
      R     #Skrajne_Prawo;
      R     #Pozycj_Warunkowe;
NETWORK
TITLE =
//Pozycjonowanie lewo
//
//
//Pozycjonowanie w lewo
      A     #i_Zez_Na_Rolki;
      A     #Pozycjonuj_Lewo;
      A     #Pozycja_Wyjsciowa;
      S     #Help_Motor_Lewo;
      S     #Help_Motor_Wolno;
      S     #Help_Poz_Lewo;
      R     #Pozycja_Srodek;
      CALL  #Tim_Jazdy_Lewo (
           IN                       := #Help_Poz_Lewo,
           STOP                     := #Stop_Bezpieczenistwa,
           PT                       := #Czas_Lewo,
           Q_0                      := #Temp_Help_2,
           ET                       := #Czas_Aktualny);
      A     #Temp_Help_2;
      O;
      AN    #Foto_Tyl;
      A     #Help_Poz_Lewo;
      S     #Pozycja_Lewo;
      S     #Potw_Pozycji;
      R     #Help_Motor_Lewo;
      R     #Help_Motor_Wolno;
      R     #Help_Poz_Lewo;
//Powrot z pozycjonowania. 
//Zjazd z fotokomorki aby zrobic ponowny najazd
      A     #Foto_Tyl;
      A     #Pozycja_Lewo;
      A     #Powrot_Poz;
      AN    #H_Powr_od_Lewo_1;
      S     #Help_Motor_Lewo;
      S     #Help_Motor_Wolno;
      S     #H_Repozycj_Lewo;
      R     #Potw_Pozycji;
//koniec zjazdu z fotokomorki
      AN    #Foto_Tyl;
      A     #H_Repozycj_Lewo;
      R     #Help_Motor_Lewo;
      R     #Help_Motor_Wolno;
      R     #H_Repozycj_Lewo;
      S     #Skrajne_Lewo;
//powrot na pozycje na srodku obrotnicy
      O     #Skrajne_Lewo;
      O(;
      A     #Powrot_Poz;
      A     #Pozycja_Lewo;
      );
      AN    #Foto_Tyl;
      S     #Help_Motor_Prawo;
      S     #Help_Motor_Wolno;
      S     #H_Powr_od_Lewo_1;
      R     #Help_Motor_Lewo;
      R     #Pozycja_Lewo;
      R     #Skrajne_Lewo;
NETWORK
TITLE =
//Okreselnie srodka
//Jazda  powrotna w strone prawa do œrodka
      A     #Foto_Przod;
      A     #H_Powr_od_Prawo_1;
      S     #H_Powr_Prawo;
      CALL  #Tim_Kon_Prawo (
           IN                       := #H_Powr_Prawo,
           STOP                     := #Stop_Bezpieczenistwa,
           PT                       := #Czas_Pow_Prawo,
           Q_0                      := #Temp_Help_2,
           ET                       := #Czas_Aktualny);
      A     #Foto_Tyl;
      A     #H_Powr_od_Lewo_1;
      S     #H_Powr_Lewo;
      CALL  #Tim_Kon_Lewo (
           IN                       := #H_Powr_Lewo,
           STOP                     := #Stop_Bezpieczenistwa,
           PT                       := #Czas_Pow_Lewo,
           Q_0                      := #Temp_Help_3,
           ET                       := #Czas_Aktualny);
//nieautoryzowane kasowanie srodka
      A     #i_Resetuj_Srodek;
      FP    #Zbocze_2;
      R     #Pozycja_Srodek;
      O     #Temp_Help_3;
      O     #Temp_Help_2;
      S     #Pozycja_Srodek;
      S     #Potw_Pozycji;
      R     #Pozycj_Warunkowe;
//zresetuj bity i pozycjonuj do srodka
      A     #Reset;
      FP    #Zbocze_1;
      S     #Pozycj_Warunkowe;
      R     #Pozycja_Srodek;
      R     #Potw_Pozycji;
      =     #Temp_Help_1;
      O     #Temp_Help_1;
      O     #Temp_Help_2;
      O     #Temp_Help_3;
      R     #Help_Motor_Prawo;
      R     #Help_Motor_Lewo;
      R     #Help_Motor_Wolno;
      R     #H_Powr_od_Prawo_1;
      R     #H_Powr_od_Lewo_1;
      R     #H_Repozycj_Prawo;
      R     #H_Repozycj_Lewo;
      R     #Help_Poz_Prawo;
      R     #Help_Poz_Lewo;
      R     #Skrajne_Prawo;
      R     #Skrajne_Lewo;
      R     #H_Powr_Prawo;
      R     #H_Powr_Lewo;
      R     #Pozycja_Prawo;
      R     #Pozycja_Lewo;
NETWORK
TITLE =
//Przyporzadkowanie wyjsc
      A     #i_Auto_Reczny;
      A     #i_Zez_Na_Rolki;
      A     #Help_Motor_Lewo;
      =     #Motor_Lewo;
      A     #i_Auto_Reczny;
      A     #i_Zez_Na_Rolki;
      A     #Help_Motor_Prawo;
      =     #Motor_Prawo;
      A     #i_Auto_Reczny;
      A     #Help_Motor_Wolno;
      =     #Motor_Wolno;
//Zezwolenie na obrot obrotnicy
      A(;
      A     #Foto_Przod;
      A     #Foto_Tyl;
      O;
      AN    #Foto_Przod;
      AN    #Foto_Tyl;
      );
      A     #Blokada_Obrotu_1;
      =     #Zez_Na_Obrot;
END_FUNCTION_BLOCK

FUNCTION_BLOCK "Poz_Band_Back"	// FB 56
//Funcja odpowiada za jazde rolek na pozycje zgodnie z rozkazem 
VERSION : 0.1
VAR_INPUT
  Stop_Bezpieczenistwa : BOOL ;
  Pozycjonuj_Lewo : BOOL ;
  Pozycjonuj_Prawo : BOOL ;
  Powrot_Poz : BOOL ;
  Foto_Przod : BOOL ;
  Foto_Tyl : BOOL ;
  Rolki_Odblokowane : BOOL ;
  Czas_Prawo : TIME ;
  Czas_Lewo : TIME ;
  Czas_Kontrolny : TIME ;
  Czas_Pow_Prawo : TIME ;
  Czas_Pow_Lewo : TIME ;
END_VAR
VAR_OUTPUT
  Potw_Pozycji : BOOL ;
  Pozycja_Lewo : BOOL ;	//Odniesienie do 0st
  Pozycja_Prawo : BOOL ;	//Odniesienie do 0st
  Pozycja_Srodek : BOOL ;
  Motor_Lewo : BOOL ;
  Motor_Prawo : BOOL ;
  Motor_Wolno : BOOL ;
  Blokuj_Obrotnice : BOOL ;
END_VAR
VAR
  Pozycja_Wyjsciowa : BOOL ;
  Tim_Jazdy_Prawo : FB 20;
  Tim_Jazdy_Lewo : FB 20;
  Tim_Kon_Prawo : FB 20;	//Timmer kontrolny prawo
  Tim_Kon_Lewo : FB 20;	//Timmer kontrolny lewo
  Help_Motor_Prawo : BOOL ;
  Help_Motor_Lewo : BOOL ;
  H_Repozycj_Prawo : BOOL ;
  H_Repozycj_Lewo : BOOL ;
  Help_Motor_Wolno : BOOL ;
  H_Powr_od_Prawo_1 : BOOL ;
  H_Powr_od_Lewo_1 : BOOL ;
  H_Powr : BOOL ;
  Help_Poz_Prawo : BOOL ;
  Help_Poz_Lewo : BOOL ;
  Pozycj_Warunkowe : BOOL ;
  Skrajne_Prawo : BOOL ;
  Skrajne_Lewo : BOOL ;
  Cykl_Norm : BOOL ;
  H4 : BOOL ;
  H5 : BOOL ;
  H6 : BOOL ;
  H7 : BOOL ;
  H8 : BOOL ;
END_VAR
VAR_TEMP
  Temp_Help_1 : BOOL ;
  Temp_Help_2 : BOOL ;
  Czas_Aktualny : TIME ;
END_VAR
BEGIN
NETWORK
TITLE =
      A     #Foto_Przod;
      A     #Foto_Tyl;
      A     #Pozycja_Srodek;
      A     #Rolki_Odblokowane;	//rolki sa odblokowane w pozycji 0st lub 180st
      =     #Pozycja_Wyjsciowa;
//warunkowe pozycjonowanie 
      O     #Pozycjonuj_Lewo;
      O     #Pozycjonuj_Prawo;
      A     #Foto_Przod;
      A     #Foto_Tyl;
      A     #Rolki_Odblokowane;
      AN    #H_Repozycj_Prawo;
      AN    #H_Powr_od_Prawo_1;
      AN    #Pozycja_Prawo;
      AN    #Pozycja_Lewo;
      AN    #Pozycja_Srodek;
      AN    #Cykl_Norm;
      S     #Pozycj_Warunkowe;
NETWORK
TITLE =
//Pozycjonowanie prawo
//Pozycjonowanie w prawo
      A     #Pozycjonuj_Prawo;
      A     #Pozycja_Wyjsciowa;
      S     #Help_Motor_Prawo;
      S     #Help_Motor_Wolno;
      S     #Help_Poz_Prawo;
      R     #Pozycja_Srodek;
      S     #Cykl_Norm;	//cykl pracy normalny
      CALL  #Tim_Jazdy_Prawo (
           IN                       := #Help_Poz_Prawo,
           STOP                     := #Stop_Bezpieczenistwa,
           PT                       := #Czas_Prawo,
           Q_0                      := #Temp_Help_2,
           ET                       := #Czas_Aktualny);
      A     #Temp_Help_2;
      O;
      A     #Help_Poz_Prawo;
      AN    #Foto_Przod;
      S     #Pozycja_Prawo;
      S     #Potw_Pozycji;
      R     #Help_Motor_Prawo;
      R     #Help_Motor_Wolno;
      R     #Help_Poz_Prawo;
//Powrot z pozycjonowania. 
//Zjazd z fotokomorki aby zrobic ponowny najazd
      O(;
      A     #Foto_Przod;
      A     #Pozycja_Prawo;
      A     #Powrot_Poz;
      AN    #H_Powr_od_Prawo_1;
      );
      O(;
      A     #Pozycj_Warunkowe;
      );
      S     #Help_Motor_Prawo;
      S     #Help_Motor_Wolno;
      S     #H_Repozycj_Prawo;
      R     #Potw_Pozycji;
      R     #Pozycja_Prawo;
//koniec zjazdu z fotokomorki
      AN    #Foto_Przod;
      A     #H_Repozycj_Prawo;
      R     #Help_Motor_Prawo;
      R     #Help_Motor_Wolno;
      R     #H_Repozycj_Prawo;
      S     #Skrajne_Prawo;
//powrot na pozycje na srodku obrtnicy
      A(;
      O     #Powrot_Poz;
      O     #Pozycj_Warunkowe;
      );
      A(;
      O     #Pozycja_Prawo;
      O     #Skrajne_Prawo;
      );
      AN    #Foto_Przod;
      S     #Help_Motor_Lewo;
      S     #Help_Motor_Wolno;
      S     #H_Powr_od_Prawo_1;
      R     #Help_Motor_Prawo;
      R     #Pozycja_Prawo;
      R     #Skrajne_Prawo;
      R     #Pozycj_Warunkowe;
NETWORK
TITLE =
//Pozycjonowanie lewo
////Pozycjonowanie w lewo
//
//      A     #Pozycjonuj_Lewo
//      A     #Pozycja_Wyjsciowa
//      S     #Help_Motor_Lewo
//      S     #Help_Motor_Wolno
//      S     #Help_Poz_Lewo
//      R     #Pozycja_Srodek
//
//      CALL  #Tim_Jazdy_Lewo
//       IN  :=#Help_Poz_Lewo
//       STOP:=#Stop_Bezpieczenistwa
//       PT  :=#Czas_Lewo
//       Q_0 :=#Temp_Help_2
//       ET  :=#Czas_Aktualny
//
//      A     #Temp_Help_2
//      O     
//      AN    #Foto_Tyl
//      A     #Help_Poz_Lewo
//      S     #Pozycja_Lewo
//      S     #Potw_Pozycji
//      R     #Help_Motor_Lewo
//      R     #Help_Motor_Wolno
//      R     #Help_Poz_Lewo
//
//
//
////Powrot z pozycjonowania. 
////Zjazd z fotokomorki aby zrobic ponowny najazd
//
//
//      A     #Foto_Tyl
//      A     #Pozycja_Lewo
//      A     #Powrot_Poz
//      AN    #H_Powr_od_Lewo_1
//      S     #Help_Motor_Lewo
//      S     #Help_Motor_Wolno
//      S     #H_Repozycj_Lewo
//      R     #Potw_Pozycji
//
//
////koniec zjazdu z fotokomorki
//
//
//      AN    #Foto_Tyl
//      A     #H_Repozycj_Lewo
//      R     #Help_Motor_Lewo
//      R     #Help_Motor_Wolno
//      R     #H_Repozycj_Lewo
//      S     #Skrajne_Lewo
//
////powrot na pozycje na srodku obrotnicy
//
//      O     #Pozycja_Lewo
//      O     #Skrajne_Lewo
//      AN    #Foto_Tyl
//      A     #Powrot_Poz
//      AN    #Help_Motor_Lewo
//      S     #Help_Motor_Prawo
//      S     #Help_Motor_Wolno
//      S     #H_Powr_od_Lewo_1
//      R     #Help_Motor_Lewo
//      R     #Pozycja_Lewo
//      R     #Skrajne_Lewo
//
NETWORK
TITLE =
//Okreselnie srodka
//Jazda  powrotna w strone prawa do œrodka
      A     #Foto_Przod;
      A     #H_Powr_od_Prawo_1;
      O;
      A     #Foto_Tyl;
      A     #H_Powr_od_Lewo_1;
      S     #H_Powr;
      CALL  #Tim_Kon_Lewo (
           IN                       := #H_Powr,
           STOP                     := #Stop_Bezpieczenistwa,
           PT                       := #Czas_Pow_Lewo,
           Q_0                      := #Temp_Help_2,
           ET                       := #Czas_Aktualny);
      A     #Temp_Help_2;
      S     #Pozycja_Srodek;
      S     #Potw_Pozycji;
      R     #Help_Motor_Prawo;
      R     #Help_Motor_Lewo;
      R     #Help_Motor_Wolno;
      R     #H_Powr_od_Prawo_1;
      R     #H_Powr_od_Lewo_1;
      R     #H_Repozycj_Prawo;
      R     #H_Repozycj_Lewo;
      R     #Help_Poz_Prawo;
      R     #Help_Poz_Lewo;
      R     #Pozycj_Warunkowe;
      R     #Skrajne_Prawo;
      R     #Skrajne_Lewo;
      R     #H_Powr;
      R     #Pozycja_Prawo;
      R     #Pozycja_Lewo;
      R     #Cykl_Norm;
      R     #Cykl_Norm;
NETWORK
TITLE =
//Przyporzadkowanie wyjsc
      A     #Help_Motor_Lewo;
      =     #Motor_Lewo;
      A     #Help_Motor_Prawo;
      =     #Motor_Prawo;
      A     #Help_Motor_Wolno;
      =     #Motor_Wolno;
END_FUNCTION_BLOCK

FUNCTION_BLOCK "Bindownica_Test"	// FB 57
VERSION : 0.1
VAR_INPUT
  i_Bind_Obwod_Ok : BOOL ;	//270 stopni
  i_Bind_Poz_Podst : BOOL ;
  i_Bind_Syg_Got : BOOL ;
  i_Bind_Blad : BOOL ;
  i_Bind_Start_Kon : BOOL ;	//Bindownica start koniec wiazania
  i_Przesznuruj : BOOL ;	//Przesznurowanie imituje bindownice
  i_Cykl_Bindowanie : BOOL ;
END_VAR
VAR_OUTPUT
  io_Bind_Obwod_Ok : BOOL ;	//270 stopni
  io_Bind_Poz_Podst : BOOL ;
  io_Bind_Syg_Got : BOOL ;
  io_Bind_Blad : BOOL ;
  io_Bind_Start_Kon : BOOL ;	//Bindownica start koniec wiazania
END_VAR
VAR
  CZas_Testowy : SFB 4;
END_VAR
VAR_TEMP
  temp_help_1 : BOOL ;
END_VAR
BEGIN
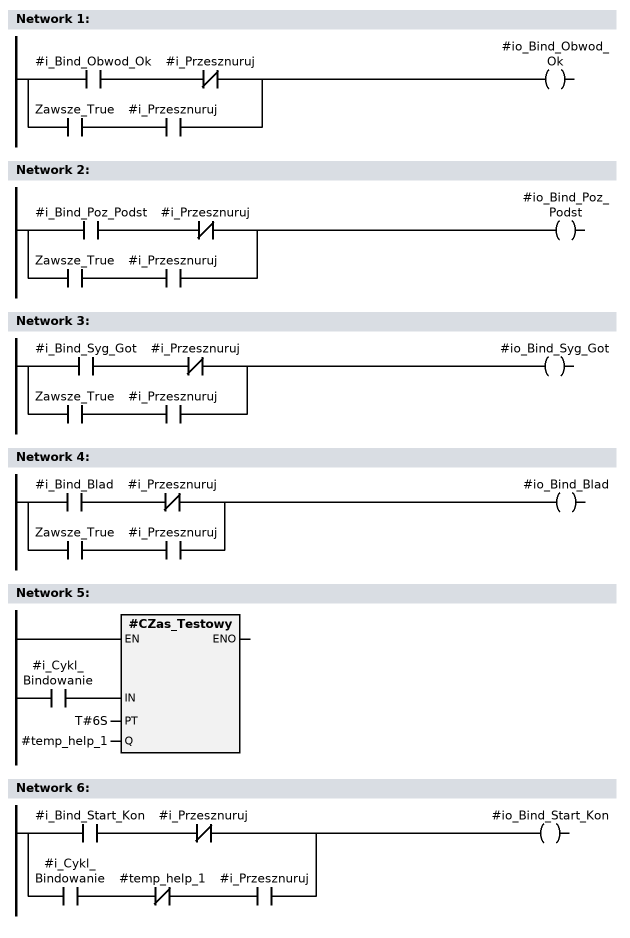
NETWORK
TITLE =
//bind obwod ok
      A     #i_Bind_Obwod_Ok;
      AN    #i_Przesznuruj;
      O;
      A     "Zawsze_True";
      A     #i_Przesznuruj;
      =     #io_Bind_Obwod_Ok;
NETWORK
TITLE =
//Pozycja podstawowa
      A     #i_Bind_Poz_Podst;
      AN    #i_Przesznuruj;
      O;
      A     "Zawsze_True";
      A     #i_Przesznuruj;
      =     #io_Bind_Poz_Podst;
NETWORK
TITLE =
//sygnal gotowosc
      A     #i_Bind_Syg_Got;
      AN    #i_Przesznuruj;
      O;
      A     "Zawsze_True";
      A     #i_Przesznuruj;
      =     #io_Bind_Syg_Got;
NETWORK
TITLE =
//Blad bindowania
      A     #i_Bind_Blad;
      AN    #i_Przesznuruj;
      O;
      A     "Zawsze_True";
      A     #i_Przesznuruj;
      =     #io_Bind_Blad;
NETWORK
TITLE =
//bindowanie
//
      A     #i_Cykl_Bindowanie;
      =     L 1.0;
      BLD   103;
      CALL  #CZas_Testowy (
           IN                       := L 1.0,
           PT                       := T#6S,
           Q                        := #temp_help_1);
      NOP   0;
NETWORK
TITLE =
//start koniec bindowania
      A     #i_Bind_Start_Kon;
      AN    #i_Przesznuruj;
      O;
      A     #i_Cykl_Bindowanie;
      AN    #temp_help_1;
      A     #i_Przesznuruj;
      =     #io_Bind_Start_Kon;
END_FUNCTION_BLOCK

FUNCTION_BLOCK "Pozycjonowanie_Palety"	// FB 58
//Funcja odpowiada za jazde rolek na pozycje zgodnie z rozkazem. Zmiany do wersji 
//porzednie:
//
//-o powrocie z pozycjonowania gdy stan pozycji palety jest nieustalony decyduje
// bit wejsciowy reset
//
VERSION : 0.1
VAR_INPUT
  i_Marka_Bezpieczenstwa : BOOL ;
  i_Rezerwa : BOOL ;
  i_Auto_Reczny : BOOL ;
  i_Pozycjonuj_Lewo : BOOL ;
  i_Pozycjonuj_Prawo : BOOL ;
  i_Pozycjonuj_Srodek : BOOL ;
  i_Foto_Przod : BOOL ;
  i_Foto_Tyl : BOOL ;
  s_i_Zez_Na_Rolki : BOOL ;
  i_Czas_Jazdy_Prawo : TIME ;
  i_Czas_Jazdy_Lewo : TIME ;
  i_Czas_Opoznienia : TIME ;
  i_Czas_Powrotu_Prawo : TIME ;
  i_Czas_Powrotu_Lewo : TIME ;
  s_i_Blokada_Obrotu : BOOL ;
  i_Resetuj_Srodek : BOOL ;	//Resetowanie zewnetrzne konca palety
  i_Setuj_Srodek : BOOL ;	//Ustawienie zewnetrzne srodka palety
END_VAR
VAR_OUTPUT
  o_Pozycja_Lewo : BOOL ;	//Odniesienie do 0st
  o_Pozycja_Prawo : BOOL ;	//Odniesienie do 0st
  o_Pozycja_Srodek : BOOL ;
  o_Potw_Pozycji : BOOL ;
  o_Motor_Lewo : BOOL ;
  o_Motor_Prawo : BOOL ;
  o_Motor_Wolno : BOOL ;
  s_o_Zez_Na_Obrot : BOOL ;
  o_Rezerwa_1 : BOOL ;
  o_Rezerwa_2 : BOOL ;
  o_Rezerwa_3 : BOOL ;
END_VAR
VAR
  Tim_Jazdy_Lewo : FB 20;
  Tim_Jazdy_Prawo : FB 20;
  Tim_Kon_Prawo : FB 20;	//Timmer kontrolny prawo
  Tim_Kon_Lewo : FB 20;	//Timmer kontrolny lewo
  Tim_Opoznienia : FB 20;
  Stop_Czas_Kontrolny : BOOL ;
  Help_Motor_Prawo : BOOL ;
  Help_Motor_Lewo : BOOL ;
  Help_Motor_Wolno : BOOL ;
  H_Repozycj_Prawo : BOOL ;
  H_Repozycj_Lewo : BOOL ;
  H_Powrot_od_Prawej : BOOL ;
  H_Powrot_od_Lewej : BOOL ;
  H_Czas_Powr_Prawo : BOOL ;
  H_Czas_Powr_Lewo : BOOL ;
  H_Czas_Jazdy_Prawo : BOOL ;
  H_Czas_Jazdy_Lewo : BOOL ;
  H_Krawedz_Prawo : BOOL ;
  H_Krawedz_Lewo : BOOL ;
  H_Pozycja_Wyjsciowa : BOOL ;
  H_Brak_Pozycji : BOOL ;
  Zbocze_1 : BOOL ;
  Zbocze_2 : BOOL ;
  H_Jakas_Pozycja : BOOL ;
  H8 : BOOL ;
  H9 : BOOL ;
  H10 : BOOL ;
  H11 : BOOL ;
  H12 : BOOL ;
END_VAR
VAR_TEMP
  Temp_Help_1 : BOOL ;
  Temp_Help_2 : BOOL ;
  Temp_Help_3 : BOOL ;
  Temp_Help_4 : BOOL ;
  Czas_Aktualny : TIME ;
END_VAR
BEGIN
NETWORK
TITLE =
//Ten network celowo ma byc wolny
NETWORK
TITLE =
//Zatrzymanie czasu w timmerach gdy obwod bezpieczenstwa nie ok
      A     #i_Marka_Bezpieczenstwa;
      S     #Stop_Czas_Kontrolny;
      AN    #i_Marka_Bezpieczenstwa;
      AN    #Stop_Czas_Kontrolny;
      JC    end;
      AN    #i_Marka_Bezpieczenstwa;
      R     #Stop_Czas_Kontrolny;
NETWORK
TITLE =
      A     #i_Foto_Przod;
      A     #i_Foto_Tyl;
      A     #o_Pozycja_Srodek;
      A     #s_i_Zez_Na_Rolki;	//rolki sa odblokowane w pozycji 0st lub 180st
      =     #H_Pozycja_Wyjsciowa;
//Reset pozycji gdy silnki wykonaja ruch
      O     #Help_Motor_Lewo;
      O     #Help_Motor_Prawo;
      R     #o_Pozycja_Prawo;
      R     #o_Pozycja_Srodek;
      R     #o_Pozycja_Lewo;
//warunkowe pozycjonowanie brak pozycji
      AN    #o_Pozycja_Prawo;
      AN    #o_Pozycja_Lewo;
      AN    #o_Pozycja_Srodek;
      =     #H_Brak_Pozycji;
      NOT;
      =     #H_Jakas_Pozycja;
NETWORK
TITLE =
//Pozycjonowanie prawo
//Pozycjonowanie w prawo
      A     #i_Pozycjonuj_Prawo;
      AN    #i_Pozycjonuj_Srodek;
      AN    #i_Pozycjonuj_Lewo;
      A     #H_Pozycja_Wyjsciowa;
      S     #Help_Motor_Prawo;
      R     #Help_Motor_Lewo;
      S     #H_Czas_Jazdy_Prawo;
//Uruchom zjazd z fotokomorki
      CALL  #Tim_Jazdy_Prawo (
           IN                       := #H_Czas_Jazdy_Prawo,
           STOP                     := #Stop_Czas_Kontrolny,
           PT                       := #i_Czas_Jazdy_Prawo,
           Q_0                      := #Temp_Help_2,
           ET                       := #Czas_Aktualny);
      A     #Temp_Help_2;
      O;
      A     #H_Czas_Jazdy_Prawo;
      AN    #i_Foto_Przod;
      S     #o_Pozycja_Prawo;
      R     #Help_Motor_Prawo;
      R     #H_Czas_Jazdy_Prawo;
NETWORK
TITLE =
//Powrot ze strony prawej
//Powrot z pozycjonowania. 
//Zjazd z fotokomorki aby zrobic ponowny najazd
      O     #o_Pozycja_Prawo;
      O     #H_Brak_Pozycji;
      A     #i_Pozycjonuj_Srodek;
      A     #i_Foto_Przod;
      A     #i_Foto_Tyl;
      A     #s_i_Zez_Na_Rolki;
      AN    #H_Powrot_od_Prawej;
      S     #Help_Motor_Prawo;
      S     #H_Repozycj_Prawo;
      R     #Help_Motor_Lewo;
//koniec zjazdu z fotokomorki
      AN    #i_Foto_Przod;
//      A     #H_Repozycj_Prawo
      R     #Help_Motor_Prawo;
      R     #H_Repozycj_Prawo;
      S     #H_Krawedz_Prawo;
//powrot na pozycje na srodku obrotnicy
      A(;
      O     #i_Pozycjonuj_Srodek;
      O     #H_Krawedz_Prawo;
      );
      A(;
      O     #o_Pozycja_Prawo;
      O     #H_Krawedz_Prawo;
      );
      AN    #i_Foto_Przod;
      S     #Help_Motor_Lewo;
      S     #H_Powrot_od_Prawej;
      R     #Help_Motor_Prawo;
      R     #H_Krawedz_Prawo;
NETWORK
TITLE =
//Pozycjonowanie lewo
//
//
//Pozycjonowanie w lewo
      A     #i_Pozycjonuj_Lewo;
      AN    #i_Pozycjonuj_Srodek;
      AN    #i_Pozycjonuj_Prawo;
      A     #H_Pozycja_Wyjsciowa;
      S     #Help_Motor_Lewo;
      R     #Help_Motor_Prawo;
      S     #H_Czas_Jazdy_Lewo;
      CALL  #Tim_Jazdy_Lewo (
           IN                       := #H_Czas_Jazdy_Lewo,
           STOP                     := #Stop_Czas_Kontrolny,
           PT                       := #i_Czas_Jazdy_Lewo,
           Q_0                      := #Temp_Help_2,
           ET                       := #Czas_Aktualny);
      A     #Temp_Help_2;
      O;
      A     #H_Czas_Jazdy_Lewo;
      AN    #i_Foto_Tyl;
      S     #o_Pozycja_Lewo;
      R     #Help_Motor_Lewo;
      R     #H_Czas_Jazdy_Lewo;
NETWORK
TITLE =
//Powrot ze strony lewej
//Powrot z pozycjonowania. 
//Zjazd z fotokomorki aby zrobic ponowny najazd
      A     #i_Pozycjonuj_Srodek;
      A     #i_Foto_Przod;
      A     #i_Foto_Tyl;
      A     #o_Pozycja_Lewo;
      A     #s_i_Zez_Na_Rolki;
      AN    #H_Powrot_od_Lewej;
      S     #Help_Motor_Lewo;
      R     #Help_Motor_Prawo;
      S     #H_Repozycj_Lewo;
//koniec zjazdu z fotokomorki
      AN    #i_Foto_Tyl;
      A     #H_Repozycj_Lewo;
      R     #Help_Motor_Lewo;
      R     #H_Repozycj_Lewo;
      S     #H_Krawedz_Lewo;
//powrot na pozycje na srodku obrotnicy
      O     #H_Krawedz_Lewo;
      O(;
      A     #i_Pozycjonuj_Srodek;
      A     #o_Pozycja_Lewo;
      );
      AN    #i_Foto_Tyl;
      S     #Help_Motor_Prawo;
      S     #H_Powrot_od_Lewej;
      R     #Help_Motor_Lewo;
      R     #H_Krawedz_Lewo;
NETWORK
TITLE =
//Okreselnie srodka
//Jazda  powrotna w strone prawa do œrodka
      A     #i_Foto_Przod;
      A     #H_Powrot_od_Prawej;
      S     #H_Czas_Powr_Prawo;
      CALL  #Tim_Kon_Prawo (
           IN                       := #H_Czas_Powr_Prawo,
           STOP                     := #Stop_Czas_Kontrolny,
           PT                       := #i_Czas_Powrotu_Prawo,
           Q_0                      := #Temp_Help_1,
           ET                       := #Czas_Aktualny);
//Powrot ze strony lewej do srodka
      A     #i_Foto_Tyl;
      A     #H_Powrot_od_Lewej;
      S     #H_Czas_Powr_Lewo;
      CALL  #Tim_Kon_Lewo (
           IN                       := #H_Czas_Powr_Lewo,
           STOP                     := #Stop_Czas_Kontrolny,
           PT                       := #i_Czas_Powrotu_Lewo,
           Q_0                      := #Temp_Help_2,
           ET                       := #Czas_Aktualny);
//nieautoryzowane kasowanie srodka
      A     #i_Resetuj_Srodek;
      R     #o_Pozycja_Srodek;
      =     #Temp_Help_3;
//nieautoryzowane setowanie  srodka
      A     #i_Setuj_Srodek;
      FP    #Zbocze_1;
      A     #i_Foto_Przod;
      A     #i_Foto_Tyl;
      S     #o_Pozycja_Srodek;
      =     #Temp_Help_4;
      O     #Temp_Help_1;
      O     #Temp_Help_2;
      S     #o_Pozycja_Srodek;
//Reset wszystkich zbedncyh bitow
      O     #Temp_Help_1;
      O     #Temp_Help_2;
      O     #Temp_Help_3;
      O     #Temp_Help_4;
      R     #Help_Motor_Prawo;
      R     #Help_Motor_Lewo;
      R     #H_Powrot_od_Prawej;
      R     #H_Powrot_od_Lewej;
      R     #H_Repozycj_Prawo;
      R     #H_Repozycj_Lewo;
      R     #H_Czas_Jazdy_Prawo;
      R     #H_Czas_Jazdy_Lewo;
      R     #H_Krawedz_Prawo;
      R     #H_Krawedz_Lewo;
      R     #H_Czas_Powr_Prawo;
      R     #H_Czas_Powr_Lewo;
      R     #o_Pozycja_Prawo;
      R     #o_Pozycja_Lewo;
NETWORK
TITLE =
//Jezeli dluzej niz 1.5 sekundy to pozycja potwierdzona
      CALL  #Tim_Opoznienia (
           IN                       := #H_Jakas_Pozycja,
           STOP                     := #Stop_Czas_Kontrolny,
           PT                       := T#1S500MS,
           Q_0                      := #o_Potw_Pozycji);
NETWORK
TITLE =
//Przyporzadkowanie wyjsc
end:  NOP   0;
//-
      A     #i_Auto_Reczny;
      A     #i_Marka_Bezpieczenstwa;
      A     #s_i_Zez_Na_Rolki;
      A     #Help_Motor_Lewo;
      AN    #Help_Motor_Prawo;
      =     #o_Motor_Lewo;
//-
      A     #i_Auto_Reczny;
      A     #i_Marka_Bezpieczenstwa;
      A     #s_i_Zez_Na_Rolki;
      A     #Help_Motor_Prawo;
      AN    #Help_Motor_Lewo;
      =     #o_Motor_Prawo;
//-
      O     #o_Motor_Lewo;
      O     #o_Motor_Prawo;
      =     #o_Motor_Wolno;
//Zezwolenie na obrot obrotnicy
      A(;
      A     #i_Foto_Przod;
      A     #i_Foto_Tyl;
      O;
      AN    #i_Foto_Przod;
      AN    #i_Foto_Tyl;
      );
      A     #s_i_Blokada_Obrotu;
      =     #s_o_Zez_Na_Obrot;
END_FUNCTION_BLOCK

FUNCTION "Funkcja_Bezpieczenstwa" : VOID	// FC 3
//Funkcja steruje bezpieczenstwem maszyny
VERSION : 0.1
VAR_TEMP
  Help_Bit : BOOL ;
END_VAR
BEGIN
NETWORK
TITLE =
//Ten Network celowo jest wolny
//
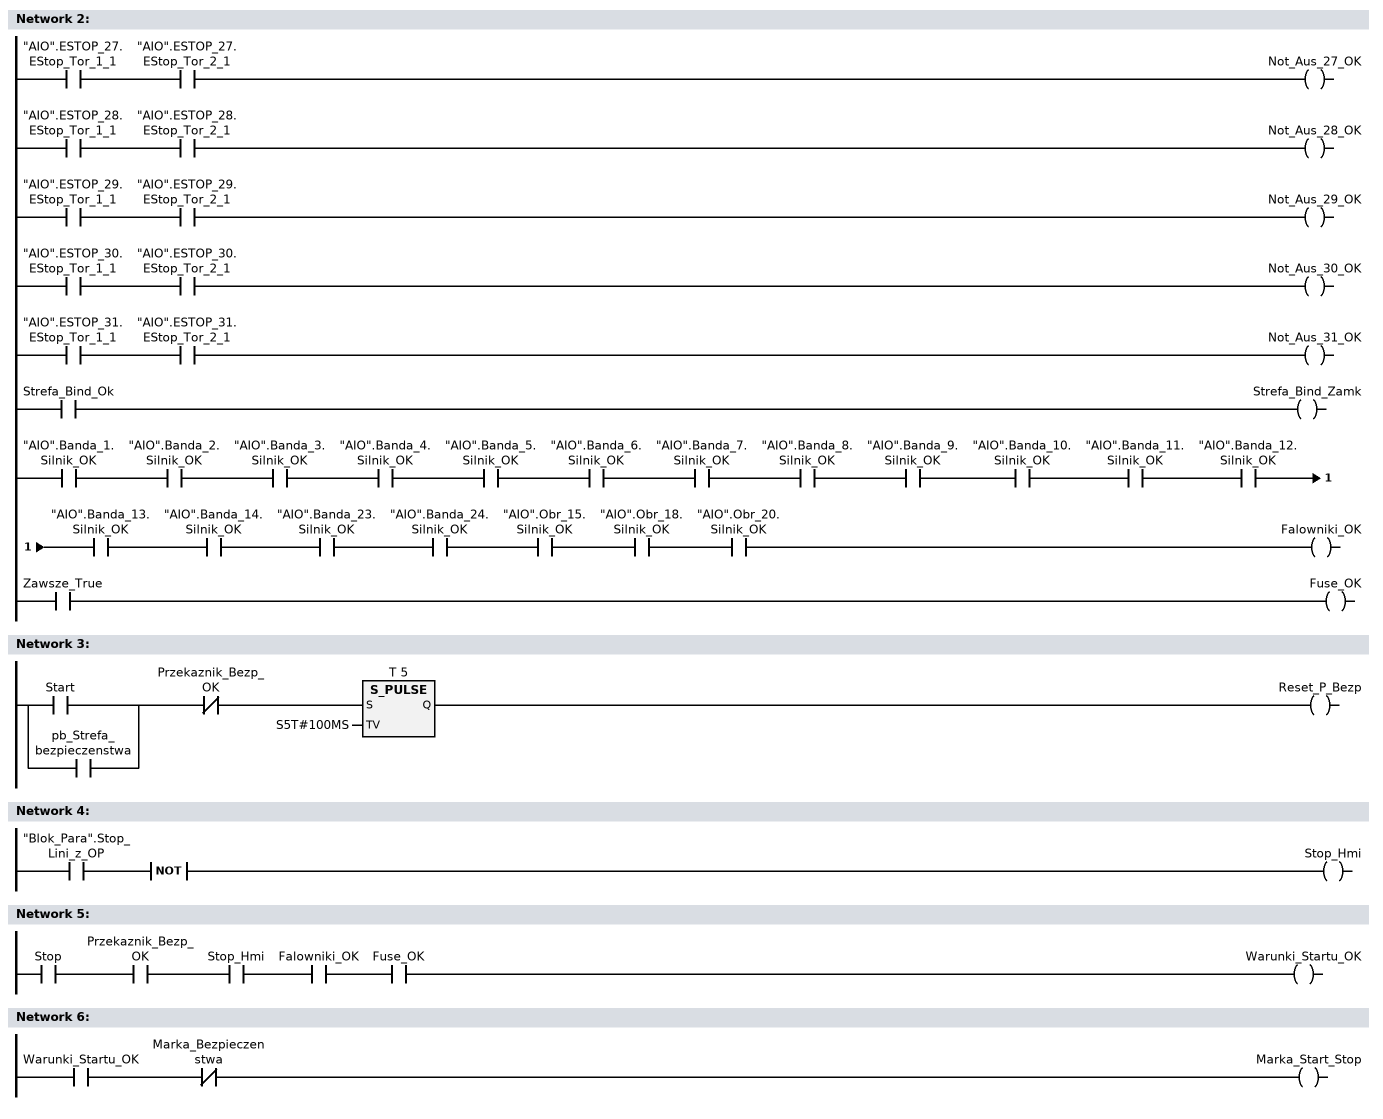
NETWORK
TITLE =
//Not Aus 27*******************************
      A     "AIO".ESTOP_27.EStop_Tor_1_1;
      A     "AIO".ESTOP_27.EStop_Tor_2_1;
      =     "Not_Aus_27_OK";
//Not Aus 28*******************************
      A     "AIO".ESTOP_28.EStop_Tor_1_1;
      A     "AIO".ESTOP_28.EStop_Tor_2_1;
      =     "Not_Aus_28_OK";
//Not Aus 29*******************************
      A     "AIO".ESTOP_29.EStop_Tor_1_1;
      A     "AIO".ESTOP_29.EStop_Tor_2_1;
      =     "Not_Aus_29_OK";
//Not Aus 30*******************************
      A     "AIO".ESTOP_30.EStop_Tor_1_1;
      A     "AIO".ESTOP_30.EStop_Tor_2_1;
      =     "Not_Aus_30_OK";
//Not Aus 31*******************************
      A     "AIO".ESTOP_31.EStop_Tor_1_1;
      A     "AIO".ESTOP_31.EStop_Tor_2_1;
      =     "Not_Aus_31_OK";
//Strefa *******************************
      A     "Strefa_Bind_Ok";
      =     "Strefa_Bind_Zamk";
//Falowniki********************************
      A     "AIO".Banda_1.Silnik_OK;
      A     "AIO".Banda_2.Silnik_OK;
      A     "AIO".Banda_3.Silnik_OK;
      A     "AIO".Banda_4.Silnik_OK;
      A     "AIO".Banda_5.Silnik_OK;
      A     "AIO".Banda_6.Silnik_OK;
      A     "AIO".Banda_7.Silnik_OK;
      A     "AIO".Banda_8.Silnik_OK;
      A     "AIO".Banda_9.Silnik_OK;
      A     "AIO".Banda_10.Silnik_OK;
      A     "AIO".Banda_11.Silnik_OK;
      A     "AIO".Banda_12.Silnik_OK;
      A     "AIO".Banda_13.Silnik_OK;
      A     "AIO".Banda_14.Silnik_OK;
      A     "AIO".Banda_23.Silnik_OK;
      A     "AIO".Banda_24.Silnik_OK;
      A     "AIO".Obr_15.Silnik_OK;
      A     "AIO".Obr_18.Silnik_OK;
      A     "AIO".Obr_20.Silnik_OK;
      =     "Falowniki_OK";
//Bezpieczniki Szafa************************
//Brak w szafie bepiecznikow z kontrola wiec
      A     "Zawsze_True";
      =     "Fuse_OK";
NETWORK
TITLE =
//Reset przekaznika bezp
      A(;
      O     "Start";
      O     "pb_Strefa_bezpieczenstwa";
      );
      AN    "Przekaznik_Bezp_OK";
      L     S5T#100MS;
      SP    T 5;
      NOP   0;
      NOP   0;
      NOP   0;
      A     T 5;
      =     "Reset_P_Bezp";
NETWORK
TITLE =
      A     "Blok_Para".Stop_Lini_z_OP;
      NOT;
      =     "Stop_Hmi";
NETWORK
TITLE =
//Warunki Startu 
      A     "Stop";
      A     "Przekaznik_Bezp_OK";
      A     "Stop_Hmi";
      A     "Falowniki_OK";
      A     "Fuse_OK";
      =     "Warunki_Startu_OK";
NETWORK
TITLE =
//warunki do strartu ok ale start nie wcisniety
      A     "Warunki_Startu_OK";
      AN    "Marka_Bezpieczenstwa";
      =     "Marka_Start_Stop";
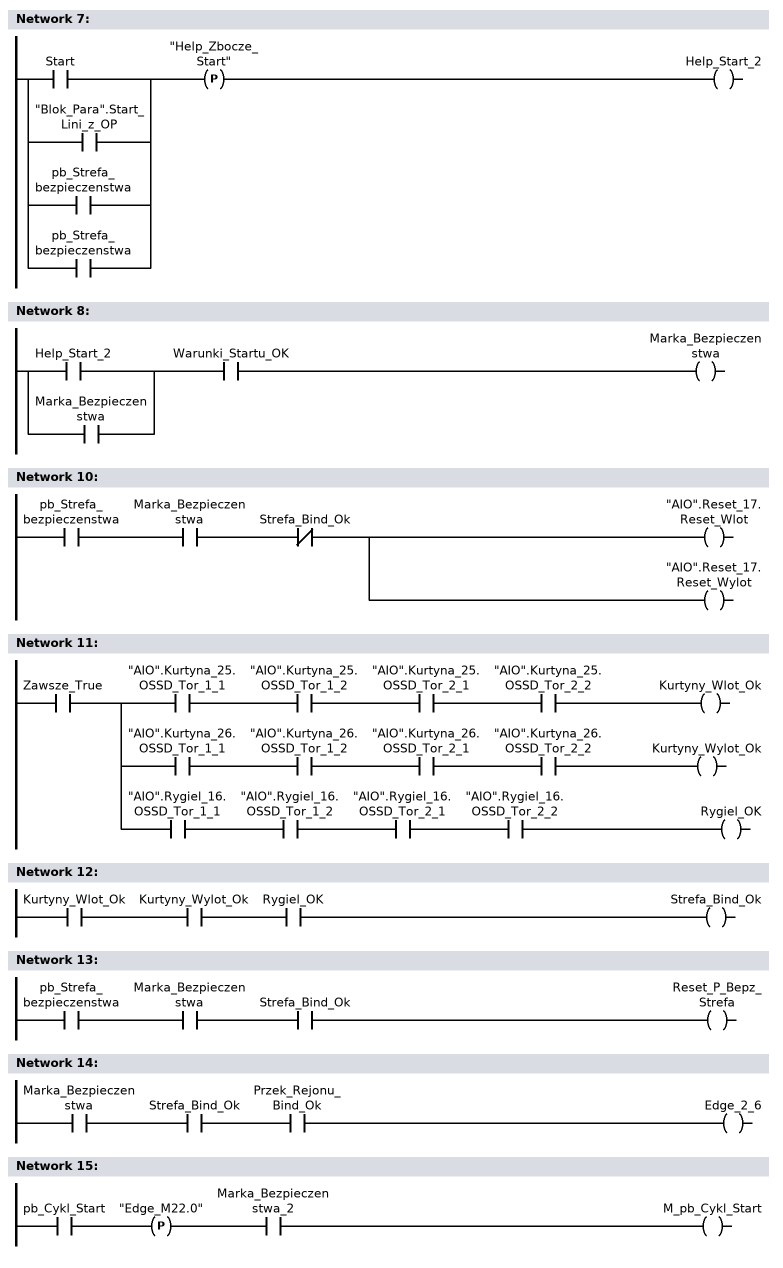
NETWORK
TITLE =
//Start na szafie glownej
      A(;
      O     "Start";
      O     "Blok_Para".Start_Lini_z_OP;
      O     "pb_Strefa_bezpieczenstwa";
      O     "pb_Strefa_bezpieczenstwa";
      );
      FP    "Help_Zbocze_Start";
      =     "Help_Start_2";
NETWORK
TITLE =
//Start Lini. Zalaczenie marki bezpieczenstwa
      A(;
      O     "Help_Start_2";
      O     "Marka_Bezpieczenstwa";
      );
      A     "Warunki_Startu_OK";
      =     "Marka_Bezpieczenstwa";
NETWORK
TITLE =
//Poczatek drugiego przekaznika bezpieczenstwa
NETWORK
TITLE =
//Resetowanie kurtyn bezpieczenstwa
//
      A     "pb_Strefa_bezpieczenstwa";
      A     "Marka_Bezpieczenstwa";
      AN    "Strefa_Bind_Ok";
      =     "AIO".Reset_17.Reset_Wlot;
      =     "AIO".Reset_17.Reset_Wylot;
NETWORK
TITLE =
//Kurtyny wlot ok modul 25
//Kurtyny wylot ok modull 26
//Rygiel adres 16 ok
      A     "Zawsze_True";
      =     L 1.0;
      A     L 1.0;
      A     "AIO".Kurtyna_25.OSSD_Tor_1_1;
      A     "AIO".Kurtyna_25.OSSD_Tor_1_2;
      A     "AIO".Kurtyna_25.OSSD_Tor_2_1;
      A     "AIO".Kurtyna_25.OSSD_Tor_2_2;
      =     "Kurtyny_Wlot_Ok";
      A     L 1.0;
      A     "AIO".Kurtyna_26.OSSD_Tor_1_1;
      A     "AIO".Kurtyna_26.OSSD_Tor_1_2;
      A     "AIO".Kurtyna_26.OSSD_Tor_2_1;
      A     "AIO".Kurtyna_26.OSSD_Tor_2_2;
      =     "Kurtyny_Wylot_Ok";
      A     L 1.0;
      A     "AIO".Rygiel_16.OSSD_Tor_1_1;
      A     "AIO".Rygiel_16.OSSD_Tor_1_2;
      A     "AIO".Rygiel_16.OSSD_Tor_2_1;
      A     "AIO".Rygiel_16.OSSD_Tor_2_2;
      =     "Rygiel_OK";
NETWORK
TITLE =
//Sprawdzenei czy strefa maszyny bindujacej bezpieczna
      A     "Kurtyny_Wlot_Ok";
      A     "Kurtyny_Wylot_Ok";
      A     "Rygiel_OK";
      =     "Strefa_Bind_Ok";
NETWORK
TITLE =
//Reset strefy bezpieczenstwa
      A     "pb_Strefa_bezpieczenstwa";
      A     "Marka_Bezpieczenstwa";
      A     "Strefa_Bind_Ok";
      =     "Reset_P_Bepz_Strefa";
NETWORK
TITLE =
//Marka do pracy dla lini bindujacej
//Uwzglednione sa warunki kurtyn
//
      A     "Marka_Bezpieczenstwa";
      A     "Strefa_Bind_Ok";
      A     "Przek_Rejonu_Bind_Ok";
      =     "Edge_2_6";
NETWORK
TITLE =
//Tak aby potwierdzic stop gdy paleta na obrotnicy
      A     "pb_Cykl_Start";
      FP    "Edge_M22.0";
      A     "Marka_Bezpieczenstwa_2";
      =     "M_pb_Cykl_Start";
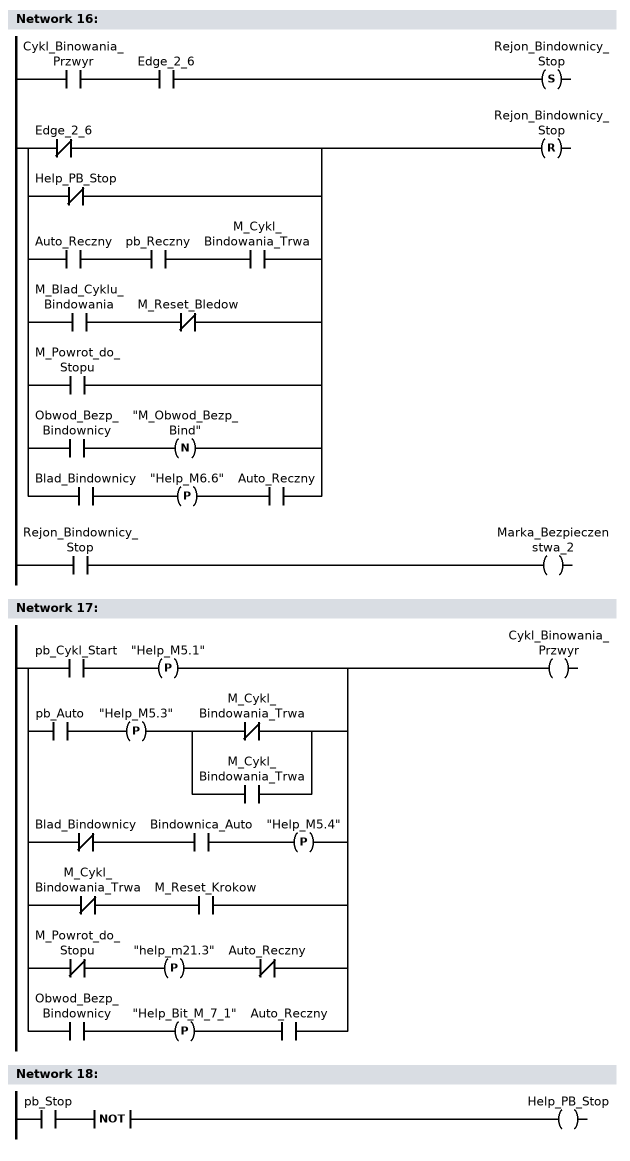
NETWORK
TITLE =
      A     "Cykl_Binowania_Przwyr";
      A     "Edge_2_6";
      S     "Rejon_Bindownicy_Stop";
      A(;
      ON    "Edge_2_6";
      ON    "Help_PB_Stop";
      O(;
      A     "Auto_Reczny";
      A     "pb_Reczny";
      A     "M_Cykl_Bindowania_Trwa";
      );
      O(;
      A     "M_Blad_Cyklu_Bindowania";
      AN    "M_Reset_Bledow";
      );
      O     "M_Powrot_do_Stopu";
      O(;
      A     "Obwod_Bezp_Bindownicy";
      FN    "M_Obwod_Bezp_Bind";
      );
      O(;
      A     "Blad_Bindownicy";
      FP    "Help_M6.6";
      A     "Auto_Reczny";
      );
      );
      R     "Rejon_Bindownicy_Stop";
      A     "Rejon_Bindownicy_Stop";
      =     "Marka_Bezpieczenstwa_2";
NETWORK
TITLE =
//Cykl bindownicy przywrocenie
//Jest wiele drog do tego samego celu 
      A     "pb_Cykl_Start";
      FP    "Help_M5.1";
      O(;
      A     "pb_Auto";
      FP    "Help_M5.3";
      A(;
      ON    "M_Cykl_Bindowania_Trwa";
      O     "M_Cykl_Bindowania_Trwa";
      );
      );
      O(;
      AN    "Blad_Bindownicy";
      A     "Bindownica_Auto";
      FP    "Help_M5.4";
      );
      O(;
      AN    "M_Cykl_Bindowania_Trwa";
      A     "M_Reset_Krokow";
      );
      O(;
      AN    "M_Powrot_do_Stopu";
      FP    "help_m21.3";
      AN    "Auto_Reczny";
      );
      O(;
      A     "Obwod_Bezp_Bindownicy";
      FP    "Help_Bit_M_7_1";
      A     "Auto_Reczny";
      );
      =     "Cykl_Binowania_Przwyr";
NETWORK
TITLE =
//Przycisk stop w automacie zatrzymuje maszyne 
      A     "pb_Stop";
      NOT;
      =     "Help_PB_Stop";
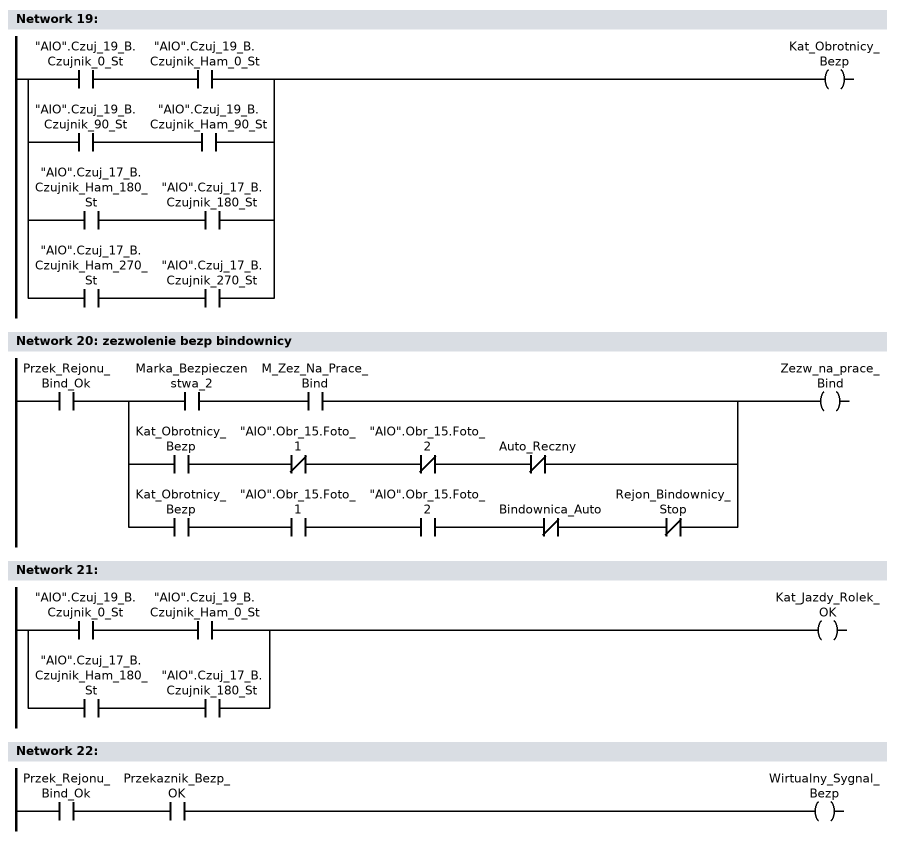
NETWORK
TITLE =
//Wysuniecie OK
      A     "AIO".Czuj_19_B.Czujnik_0_St;
      A     "AIO".Czuj_19_B.Czujnik_Ham_0_St;
      O;
      A     "AIO".Czuj_19_B.Czujnik_90_St;
      A     "AIO".Czuj_19_B.Czujnik_Ham_90_St;
      O;
      A     "AIO".Czuj_17_B.Czujnik_Ham_180_St;
      A     "AIO".Czuj_17_B.Czujnik_180_St;
      O;
      A     "AIO".Czuj_17_B.Czujnik_Ham_270_St;
      A     "AIO".Czuj_17_B.Czujnik_270_St;
      =     "Kat_Obrotnicy_Bezp";
NETWORK
TITLE = zezwolenie bezp bindownicy
//Obwod bezpieczenstwa do bindownicy.
      A     "Przek_Rejonu_Bind_Ok";
      A(;
      A     "Marka_Bezpieczenstwa_2";
      A     "M_Zez_Na_Prace_Bind";
      O;
      A     "Kat_Obrotnicy_Bezp";
      AN    "AIO".Obr_15.Foto_1;
      AN    "AIO".Obr_15.Foto_2;
      AN    "Auto_Reczny";
      O;
      A     "Kat_Obrotnicy_Bezp";
      A     "AIO".Obr_15.Foto_1;
      A     "AIO".Obr_15.Foto_2;
      AN    "Bindownica_Auto";
      AN    "Rejon_Bindownicy_Stop";
      );
      =     "Zezw_na_prace_Bind";
NETWORK
TITLE =
//Kat jazdy rolek ok 
      A     "AIO".Czuj_19_B.Czujnik_0_St;
      A     "AIO".Czuj_19_B.Czujnik_Ham_0_St;
      O;
      A     "AIO".Czuj_17_B.Czujnik_Ham_180_St;
      A     "AIO".Czuj_17_B.Czujnik_180_St;
      =     "Kat_Jazdy_Rolek_OK";
NETWORK
TITLE =
//Sygnal imitujacy kurtyne i grzyba 
      A     "Przek_Rejonu_Bind_Ok";
      A     "Przekaznik_Bezp_OK";
      =     "Wirtualny_Sygnal_Bezp";
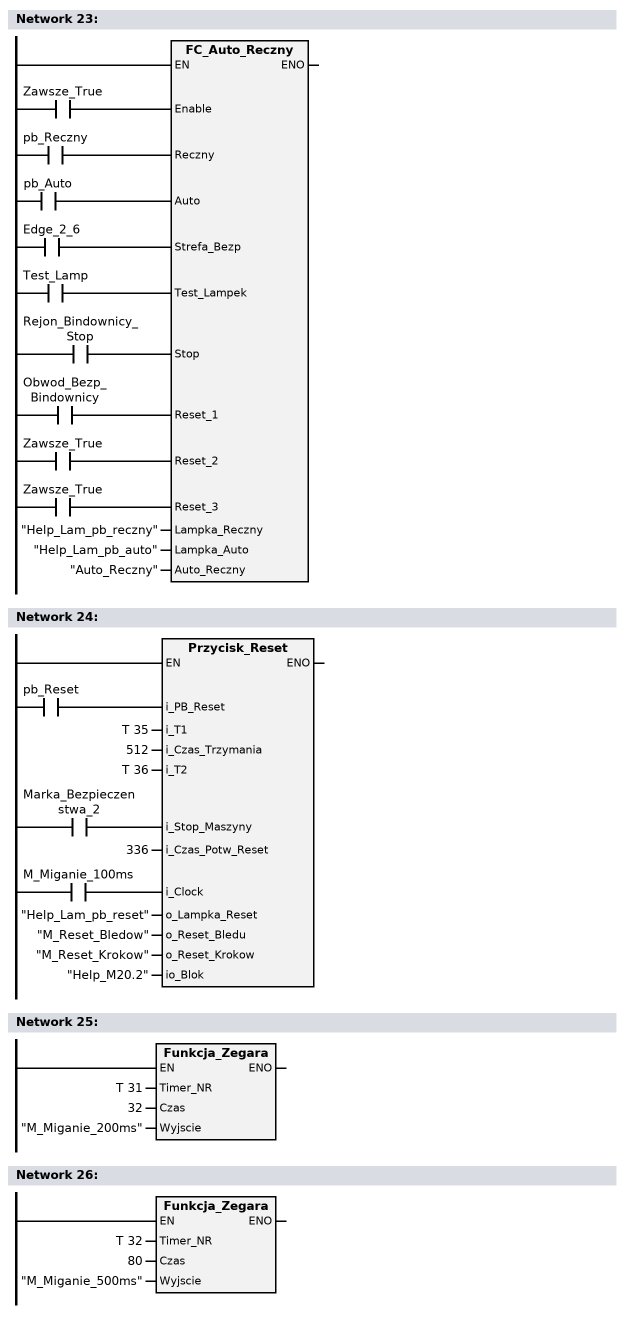
NETWORK
TITLE =
//Wybranie trybu pracy bindownicy (reczny/auto)
//Jezeli cos nie tak ze strefa to przejscie na reczny
      A     "Zawsze_True";
      =     L 1.0;
      BLD   103;
      A     "pb_Reczny";
      =     L 1.1;
      BLD   103;
      A     "pb_Auto";
      =     L 1.2;
      BLD   103;
      A     "Edge_2_6";
      =     L 1.3;
      BLD   103;
      A     "Test_Lamp";
      =     L 1.4;
      BLD   103;
      A     "Rejon_Bindownicy_Stop";
      =     L 1.5;
      BLD   103;
      A     "Obwod_Bezp_Bindownicy";
      =     L 1.6;
      BLD   103;
      A     "Zawsze_True";
      =     L 1.7;
      BLD   103;
      A     "Zawsze_True";
      =     L 2.0;
      BLD   103;
      CALL  "FC_Auto_Reczny" (
           Enable                   := L 1.0,
           Reczny                   := L 1.1,
           Auto                     := L 1.2,
           Strefa_Bezp              := L 1.3,
           Test_Lampek              := L 1.4,
           Stop                     := L 1.5,
           Reset_1                  := L 1.6,
           Reset_2                  := L 1.7,
           Reset_3                  := L 2.0,
           Lampka_Reczny            := "Help_Lam_pb_reczny",
           Lampka_Auto              := "Help_Lam_pb_auto",
           Auto_Reczny              := "Auto_Reczny");
      NOP   0;
NETWORK
TITLE =
      A     "pb_Reset";
      =     L 1.0;
      BLD   103;
      A     "Marka_Bezpieczenstwa_2";
      =     L 1.1;
      BLD   103;
      A     "M_Miganie_100ms";
      =     L 1.2;
      BLD   103;
      CALL  "Przycisk_Reset" (
           i_PB_Reset               := L 1.0,
           i_T1                     := T 35,
           i_Czas_Trzymania         := 512,
           i_T2                     := T 36,
           i_Stop_Maszyny           := L 1.1,
           i_Czas_Potw_Reset        := 336,
           i_Clock                  := L 1.2,
           o_Lampka_Reset           := "Help_Lam_pb_reset",
           o_Reset_Bledu            := "M_Reset_Bledow",
           o_Reset_Krokow           := "M_Reset_Krokow",
           io_Blok                  := "Help_M20.2");
      NOP   0;
NETWORK
TITLE =
//Timmer generujacy takt 200ms
//
      CALL  "Funkcja_Zegara" (
           Timer_NR                 := T 31,
           Czas                     := 32,
           Wyjscie                  := "M_Miganie_200ms");
      NOP   0;
NETWORK
TITLE =
//Timmer generujacy takt 500ms
      CALL  "Funkcja_Zegara" (
           Timer_NR                 := T 32,
           Czas                     := 80,
           Wyjscie                  := "M_Miganie_500ms");
      NOP   0;
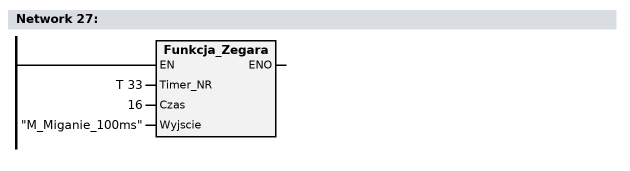
NETWORK
TITLE =
//Timmer generujacy takt 100ms
      CALL  "Funkcja_Zegara" (
           Timer_NR                 := T 33,
           Czas                     := 16,
           Wyjscie                  := "M_Miganie_100ms");
      NOP   0;
END_FUNCTION

FUNCTION "Sprawdzenie_Czujnikow" : VOID	// FC 4
VERSION : 0.1
VAR_TEMP
  Help_Zmiana_1 : BOOL ;
  Help_Zmiana_2 : BOOL ;
  Help_Zmiana_3 : BOOL ;
  Help_Zmiana_4 : BOOL ;
END_VAR
BEGIN
NETWORK
TITLE =
//Ten Network celowo wolny
NETWORK
TITLE =
//Wyznaczenie zmian
//      A     "AIO".Banda_1.Foto_1
//      =     M    400.0
//      A     "AIO".Banda_2.Foto_1
//      =     M    400.1
      A     "AIO".Banda_3.Foto_1;
      =     M 400.2;
      A     "AIO".Banda_4.Foto_1;
      =     M 400.3;
      A     "AIO".Banda_4.Foto_2;
      =     M 400.4;
      A     "AIO".Banda_5.Foto_1;
      =     M 400.5;
      A     "AIO".Banda_6.Foto_1;
      =     M 400.6;
      A     "AIO".Banda_7.Foto_1;
      =     M 400.7;
      A     "AIO".Banda_8.Foto_1;
      =     M 401.0;
      A     "AIO".Banda_9.Foto_1;
      =     M 401.1;
      A     "AIO".Banda_10.Foto_1;
      =     M 401.2;
      A     "AIO".Banda_11.Foto_1;
      =     M 401.3;
      A     "AIO".Banda_12.Foto_1;
      =     M 401.4;
      A     "AIO".Banda_13.Foto_1;
      =     M 401.5;
      A     "AIO".Banda_13.Foto_2;
      =     M 401.6;
      A     "AIO".Banda_14.Foto_1;
      =     M 401.7;
      A     "AIO".Czuj_19.Czujnik_0_St;
      =     M 402.0;
      A     "AIO".Czuj_19.Czujnik_Ham_0_St;
      =     M 402.1;
      A     "AIO".Czuj_19.Czujnik_Ham_90_St;
      =     M 402.2;
      A     "AIO".Czuj_19.Czujnik_90_St;
      =     M 402.3;
      A     "AIO".Czuj_21.Czujnik_0_St;
      =     M 402.4;
      A     "AIO".Czuj_21.Czujnik_Ham_0_St;
      =     M 22.5;
      A     "AIO".Czuj_21.Czujnik_Ham_90_St;
      =     M 402.6;
      A     "AIO".Czuj_21.Czujnik_90_St;
      =     M 402.7;
      A     "AIO".Czuj_22.Czujnik_45_St_CW;
      =     M 403.0;
      A     "AIO".Czuj_22.Czujnik_45_St_CCW;
      =     M 403.1;
      A     "AIO".Banda_10.Foto_2;
      =     M 403.2;
//Czujnik od czesci bindujacej
      A     "AIO".Banda_23.Foto_1;
      =     M 408.0;
      A     "AIO".Banda_23.Foto_2;
      =     M 408.1;
      A     "AIO".Banda_24.Foto_1;
      =     M 408.2;
      A     "AIO".Banda_24.Foto_2;
      =     M 408.3;
      A     "AIO".Banda_2.Foto_1;
      =     M 408.4;
      A     "AIO".Banda_2.Foto_2;
      =     M 408.5;
//banda 1 wyjatkowo nie ma fotokomorek
//zamiast niej ma obrotnica 15
      A     "AIO".Obr_15.Foto_1;
      =     M 408.6;
      A     "AIO".Obr_15.Foto_2;
      =     M 408.7;
//-
      A     "AIO".Czuj_19_B.Czujnik_0_St;
      =     M 409.0;
      A     "AIO".Czuj_19_B.Czujnik_Ham_0_St;
      =     M 409.1;
      A     "AIO".Czuj_19_B.Czujnik_Ham_90_St;
      =     M 409.2;
      A     "AIO".Czuj_19_B.Czujnik_90_St;
      =     M 409.3;
//-
      A     "AIO".Czuj_17_B.Czujnik_180_St;
      =     M 409.4;
      A     "AIO".Czuj_17_B.Czujnik_Ham_180_St;
      =     M 409.5;
      A     "AIO".Czuj_17_B.Czujnik_Ham_270_St;
      =     M 409.6;
      A     "AIO".Czuj_17_B.Czujnik_270_St;
      =     M 409.7;
      A     "Foto_Wozek";
      =     M 410.0;
NETWORK
TITLE =
//pierwsze 32 bity do porownania
      CALL  "Szukaj_Zmiany_2" (
           DWORD_IN_NEW             := "Nowe_Slowo_1",
           CHANGE                   := #Help_Zmiana_1,
           DWORD_IN_OLD             := "Stare_Slowo_1");
NETWORK
TITLE =
//drugie 32 bity do porownania
      CALL  "Szukaj_Zmiany_2" (
           DWORD_IN_NEW             := "Nowe_Slowo_2",
           CHANGE                   := #Help_Zmiana_2,
           DWORD_IN_OLD             := "Stare_Slowo_2");
NETWORK
TITLE =
      CALL  "Toggle" (
           Wyzwolenie_1             := #Help_Zmiana_1,
           Wyzwolenie_2             := #Help_Zmiana_2,
           Wyzwolenie_3             := "Zawsze_False",
           Wyzwolenie_4             := "Zawsze_False",
           TOGGLE                   := "Zmiana_Wykryta");
NETWORK
TITLE =
      A     "Zmiana_Wykryta";
      =     "Help_Lam_Biala";
END_FUNCTION

